C05443=1054.206,-122.391,-64.552,170.361,28.677,155.442
C05444=1054.213,-122.141,-64.561,170.364,28.677,155.442
C05445=1054.219,-121.892,-64.571,170.366,28.678,155.442
C05446=1054.225,-121.642,-64.580,170.368,28.678,155.442
C05447=1054.231,-121.393,-64.590,170.370,28.678,155.441
C05448=1054.237,-121.142,-64.598,170.371,28.679,155.441
C05449=1054.243,-120.892,-64.608,170.373,28.679,155.441
C05450=1054.249,-120.643,-64.618,170.376,28.680,155.441
C05451=1054.256,-120.393,-64.627,170.378,28.680,155.441
C05452=1054.263,-120.143,-64.636,170.380,28.681,155.441
C05453=1054.268,-119.894,-64.645,170.382,28.681,155.441
C05454=1054.274,-119.644,-64.655,170.384,28.682,155.441
C05455=1054.280,-119.394,-64.664,170.386,28.683,155.441
C05456=1054.286,-119.144,-64.673,170.389,28.683,155.441
C05457=1054.292,-118.894,-64.683,170.390,28.684,155.441
C05458=1054.299,-118.645,-64.692,170.392,28.684,155.441
C05459=1054.305,-118.395,-64.702,170.394,28.685,155.441
C05460=1054.311,-118.145,-64.712,170.396,28.685,155.440
C05461=1054.317,-117.896,-64.720,170.398,28.686,155.440
C05462=1054.323,-117.646,-64.730,170.401,28.686,155.440
C05463=1054.330,-117.397,-64.739,170.403,28.687,155.440
C05464=1054.336,-117.147,-64.749,170.405,28.688,155.440
C05465=1054.342,-116.897,-64.758,170.407,28.688,155.440
C05466=1054.348,-116.647,-64.768,170.409,28.689,155.440
C05467=1054.354,-116.397,-64.778,170.410,28.689,155.440
C05468=1054.360,-116.148,-64.787,170.412,28.689,155.440
C05469=1054.367,-115.898,-64.797,170.415,28.691,155.440
C05470=1054.373,-115.648,-64.806,170.417,28.691,155.440
C05471=1054.379,-115.364,-64.817,170.419,28.692,155.440
C05472=1054.387,-115.080,-64.828,170.422,28.692,155.440
C05473=1054.393,-114.795,-64.838,170.424,28.693,155.440
C05474=1054.401,-114.511,-64.850,170.427,28.694,155.439
C05475=1054.407,-114.261,-64.859,170.428,28.694,155.439
C05476=1054.413,-114.011,-64.869,170.430,28.695,155.439
C05477=1054.419,-113.762,-64.878,170.432,28.696,155.439
C05478=1054.425,-113.512,-64.887,170.434,28.696,155.439
C05479=1054.431,-113.263,-64.897,170.436,28.697,155.439
C05480=1054.437,-113.013,-64.908,170.439,28.698,155.439
C05481=1054.443,-112.763,-64.917,170.441,28.698,155.439
C05482=1054.449,-112.514,-64.927,170.443,28.699,155.439
C05483=1054.455,-112.264,-64.937,170.445,28.699,155.439
C05484=1054.462,-112.014,-64.946,170.446,28.700,155.439
C05485=1054.468,-111.764,-64.956,170.448,28.701,155.439
C05486=1054.474,-111.514,-64.965,170.450,28.702,155.439
C05487=1054.480,-111.265,-64.975,170.453,28.702,155.439
C05488=1054.487,-111.015,-64.985,170.455,28.703,155.439
C05489=1054.493,-110.766,-64.995,170.457,28.704,155.439
C05490=1054.498,-110.515,-65.005,170.459,28.704,155.439
C05491=1054.504,-110.266,-65.014,170.461,28.705,155.439
C05492=1054.511,-110.016,-65.024,170.462,28.706,155.439
C05493=1054.517,-109.766,-65.034,170.465,28.706,155.438
C05494=1054.523,-109.517,-65.044,170.467,28.707,155.438
C05495=1054.529,-109.267,-65.053,170.469,28.708,155.438
C05496=1054.535,-109.017,-65.063,170.471,28.708,155.438
C05497=1054.542,-108.768,-65.073,170.473,28.709,155.438
C05498=1054.548,-108.518,-65.083,170.475,28.710,155.438
C05499=1054.554,-108.268,-65.093,170.477,28.711,155.438
C05500=1054.560,-108.018,-65.103,170.479,28.711,155.438
C05501=1054.567,-107.768,-65.112,170.481,28.712,155.438
C05502=1054.573,-107.519,-65.123,170.483,28.713,155.438
C05503=1054.579,-107.269,-65.132,170.485,28.713,155.438
C05504=1054.585,-107.019,-65.142,170.487,28.714,155.438
C05505=1054.591,-106.769,-65.152,170.489,28.715,155.438
C05506=1054.597,-106.520,-65.162,170.491,28.716,155.438
C05507=1054.603,-106.270,-65.172,170.494,28.716,155.438
C05508=1054.610,-106.020,-65.181,170.495,28.717,155.438
C05509=1054.615,-105.771,-65.192,170.497,28.719,155.438
C05510=1054.622,-105.521,-65.202,170.499,28.719,155.438
C05511=1054.628,-105.271,-65.211,170.501,28.720,155.438
C05512=1054.634,-105.022,-65.222,170.503,28.720,155.438
C05513=1054.640,-104.772,-65.232,170.505,28.721,155.438
C05514=1054.646,-104.521,-65.242,170.508,28.722,155.438
C05515=1054.653,-104.272,-65.252,170.509,28.723,155.438
C05516=1054.658,-104.022,-65.262,170.511,28.724,155.438
C05517=1054.665,-103.773,-65.273,170.513,28.725,155.438
C05518=1054.671,-103.523,-65.282,170.515,28.726,155.438
C05519=1054.677,-103.273,-65.292,170.517,28.726,155.438
C05520=1054.683,-103.024,-65.303,170.519,28.727,155.438
C05521=1054.689,-102.774,-65.312,170.522,28.728,155.438
C05522=1054.695,-102.525,-65.322,170.523,28.729,155.438
C05523=1054.702,-102.274,-65.333,170.525,28.730,155.438
C05524=1054.708,-102.025,-65.343,170.527,28.731,155.438
C05525=1054.714,-101.775,-65.353,170.529,28.731,155.438
C05526=1054.720,-101.525,-65.363,170.531,28.732,155.438
C05527=1054.726,-101.276,-65.373,170.533,28.733,155.438
C05528=1054.732,-101.026,-65.383,170.536,28.734,155.437
C05529=1054.738,-100.777,-65.394,170.537,28.735,155.438
C05530=1054.745,-100.526,-65.404,170.539,28.736,155.438
C05531=1054.751,-100.277,-65.414,170.541,28.737,155.437
C05532=1054.757,-100.027,-65.424,170.543,28.738,155.437
C05533=1054.763,-99.778,-65.434,170.545,28.739,155.438
C05534=1054.769,-99.527,-65.445,170.547,28.739,155.437
C05535=1054.777,-99.242,-65.456,170.550,28.740,155.437
C05536=1054.784,-98.956,-65.468,170.551,28.741,155.437
C05537=1054.791,-98.670,-65.479,170.554,28.743,155.437
C05538=1054.798,-98.385,-65.492,170.556,28.744,155.437
C05539=1054.803,-98.135,-65.502,170.558,28.744,155.437
C05540=1054.810,-97.886,-65.512,170.560,28.745,155.437
C05541=1054.816,-97.636,-65.522,170.563,28.746,155.437
C05542=1054.822,-97.386,-65.533,170.564,28.747,155.437
C05543=1054.829,-97.137,-65.543,170.566,28.748,155.437
C05544=1054.834,-96.887,-65.553,170.568,28.749,155.437
C05545=1054.840,-96.637,-65.564,170.570,28.750,155.437
C05546=1054.847,-96.388,-65.575,170.572,28.751,155.437
C05547=1054.852,-96.138,-65.585,170.574,28.752,155.438
C05548=1054.859,-95.888,-65.595,170.575,28.753,155.438
C05549=1054.865,-95.638,-65.606,170.578,28.754,155.438
C05550=1054.871,-95.389,-65.616,170.580,28.755,155.438
C05551=1054.877,-95.139,-65.627,170.582,28.756,155.438
C05552=1054.882,-94.890,-65.638,170.584,28.757,155.438
C05553=1054.889,-94.639,-65.648,170.586,28.758,155.438
C05554=1054.895,-94.390,-65.658,170.587,28.759,155.438
C05555=1054.901,-94.140,-65.669,170.589,28.760,155.438
C05556=1054.907,-93.890,-65.679,170.591,28.761,155.438
C05557=1054.913,-93.641,-65.690,170.594,28.763,155.438
C05558=1054.920,-93.391,-65.700,170.596,28.763,155.438
C05559=1054.925,-93.141,-65.711,170.598,28.764,155.438
C05560=1054.932,-92.892,-65.721,170.600,28.765,155.438
C05561=1054.937,-92.642,-65.732,170.601,28.766,155.438
C05562=1054.944,-92.392,-65.743,170.603,28.767,155.438
C05563=1054.950,-92.143,-65.753,170.605,28.768,155.438
C05564=1054.956,-91.893,-65.763,170.607,28.769,155.438
C05565=1054.961,-91.643,-65.774,170.610,28.771,155.438
C05566=1054.968,-91.393,-65.785,170.611,28.772,155.438
C05567=1054.974,-91.144,-65.796,170.613,28.773,155.438
C05568=1054.981,-90.895,-65.806,170.615,28.774,155.438
C05569=1054.987,-90.644,-65.817,170.617,28.775,155.438
C05570=1054.992,-90.394,-65.827,170.619,28.776,155.438
C05571=1054.999,-90.145,-65.838,170.621,28.777,155.438
C05572=1055.005,-89.895,-65.849,170.622,28.778,155.438
C05573=1055.011,-89.645,-65.860,170.624,28.780,155.438
C05574=1055.017,-89.396,-65.870,170.627,28.781,155.438
C05575=1055.024,-89.146,-65.881,170.629,28.782,155.438
C05576=1055.029,-88.896,-65.892,170.631,28.783,155.438
C05577=1055.036,-88.647,-65.902,170.633,28.784,155.438
C05578=1055.041,-88.397,-65.913,170.634,28.785,155.438
C05579=1055.048,-88.147,-65.924,170.636,28.786,155.438
C05580=1055.054,-87.898,-65.934,170.638,28.787,155.438
C05581=1055.061,-87.648,-65.945,170.640,28.788,155.438
C05582=1055.066,-87.398,-65.956,170.643,28.789,155.438
C05583=1055.073,-87.149,-65.967,170.645,28.790,155.438
C05584=1055.079,-86.899,-65.978,170.646,28.791,155.439
C05585=1055.085,-86.649,-65.989,170.648,28.792,155.439
C05586=1055.091,-86.400,-65.999,170.650,28.794,155.439
C05587=1055.098,-86.150,-66.010,170.652,28.795,155.439
C05588=1055.103,-85.901,-66.021,170.654,28.796,155.439
C05589=1055.111,-85.651,-66.032,170.656,28.797,155.439
C05590=1055.116,-85.401,-66.043,170.657,28.798,155.439
C05591=1055.122,-85.152,-66.054,170.660,28.799,155.439
C05592=1055.129,-84.902,-66.064,170.662,28.800,155.439
C05593=1055.135,-84.652,-66.075,170.664,28.801,155.439
C05594=1055.141,-84.402,-66.086,170.666,28.803,155.439
C05595=1055.147,-84.153,-66.097,170.667,28.804,155.439
C05596=1055.153,-83.903,-66.108,170.669,28.805,155.439
C05597=1055.160,-83.653,-66.119,170.671,28.806,155.439
C05598=1055.165,-83.404,-66.130,170.673,28.807,155.439
C05599=1055.173,-83.120,-66.142,170.676,28.808,155.439
C05600=1055.180,-82.837,-66.154,170.678,28.810,155.439
C05601=1055.187,-82.553,-66.167,170.680,28.811,155.439
C05602=1055.194,-82.270,-66.179,170.682,28.812,155.439
C05603=1055.201,-82.020,-66.190,170.684,28.814,155.439
C05604=1055.206,-81.771,-66.201,170.686,28.815,155.440
C05605=1055.213,-81.521,-66.212,170.688,28.816,155.440
C05606=1055.219,-81.271,-66.223,170.689,28.817,155.440
C05607=1055.225,-81.021,-66.234,170.691,28.818,155.440
C05608=1055.231,-80.772,-66.245,170.694,28.820,155.440
C05609=1055.238,-80.522,-66.255,170.696,28.821,155.440
C05610=1055.244,-80.273,-66.267,170.698,28.822,155.440
C05611=1055.251,-80.023,-66.278,170.700,28.823,155.440
C05612=1055.256,-79.773,-66.289,170.701,28.825,155.440
C05613=1055.263,-79.523,-66.300,170.703,28.826,155.440
C05614=1055.269,-79.274,-66.311,170.705,28.827,155.440
C05615=1055.276,-79.024,-66.322,170.707,28.828,155.440
C05616=1055.282,-78.775,-66.334,170.709,28.829,155.440
C05617=1055.288,-78.525,-66.345,170.710,28.830,155.440
C05618=1055.294,-78.275,-66.356,170.713,28.832,155.440
C05619=1055.300,-78.025,-66.367,170.715,28.833,155.440
C05620=1055.306,-77.776,-66.378,170.717,28.835,155.441
C05621=1055.312,-77.526,-66.390,170.719,28.836,155.441
C05622=1055.318,-77.276,-66.401,170.720,28.837,155.441
C05623=1055.324,-77.026,-66.412,170.722,28.839,155.441
C05624=1055.331,-76.777,-66.423,170.724,28.840,155.441
C05625=1055.337,-76.527,-66.435,170.726,28.841,155.441
C05626=1055.343,-76.278,-66.446,170.728,28.842,155.441
C05627=1055.349,-76.027,-66.457,170.730,28.843,155.441
C05628=1055.355,-75.779,-66.468,170.731,28.845,155.441
C05629=1055.361,-75.528,-66.480,170.734,28.846,155.441
C05630=1055.367,-75.279,-66.491,170.736,28.848,155.441
C05631=1055.374,-75.029,-66.502,170.738,28.849,155.441
C05632=1055.379,-74.780,-66.513,170.739,28.851,155.441
C05633=1055.386,-74.530,-66.525,170.741,28.852,155.442
C05634=1055.392,-74.281,-66.536,170.743,28.853,155.442
C05635=1055.398,-74.031,-66.547,170.745,28.854,155.442
C05636=1055.405,-73.780,-66.559,170.747,28.856,155.442
C05637=1055.411,-73.532,-66.570,170.749,28.857,155.442
C05638=1055.417,-73.281,-66.582,170.750,28.859,155.442
C05639=1055.422,-73.032,-66.594,170.752,28.860,155.442
C05640=1055.429,-72.782,-66.605,170.754,28.861,155.442
C05641=1055.435,-72.533,-66.617,170.757,28.863,155.442
C05642=1055.441,-72.283,-66.628,170.758,28.864,155.442
C05643=1055.447,-72.033,-66.639,170.760,28.866,155.442
C05644=1055.453,-71.784,-66.651,170.762,28.867,155.443
C05645=1055.458,-71.534,-66.662,170.764,28.868,155.443
C05646=1055.465,-71.284,-66.674,170.766,28.870,155.443
C05647=1055.471,-71.035,-66.685,170.767,28.872,155.443
C05648=1055.477,-70.785,-66.697,170.769,28.873,155.443
C05649=1055.482,-70.536,-66.708,170.771,28.874,155.443
C05650=1055.489,-70.286,-66.720,170.773,28.876,155.443
C05651=1055.495,-70.036,-66.732,170.775,28.877,155.443
C05652=1055.501,-69.787,-66.744,170.776,28.879,155.443
C05653=1055.507,-69.536,-66.755,170.778,28.880,155.444
C05654=1055.513,-69.288,-66.767,170.780,28.881,155.444
C05655=1055.519,-69.037,-66.778,170.783,28.883,155.444
C05656=1055.525,-68.788,-66.790,170.784,28.885,155.444
C05657=1055.531,-68.538,-66.801,170.786,28.886,155.444
C05658=1055.538,-68.288,-66.813,170.788,28.887,155.444
C05659=1055.544,-68.040,-66.825,170.790,28.889,155.444
C05660=1055.549,-67.789,-66.837,170.792,28.891,155.444
C05661=1055.556,-67.540,-66.849,170.793,28.892,155.444
C05662=1055.562,-67.290,-66.859,170.795,28.893,155.445
C05663=1055.568,-67.009,-66.873,170.797,28.895,155.445
C05664=1055.576,-66.728,-66.886,170.800,28.897,155.445
C05665=1055.583,-66.446,-66.900,170.801,28.898,155.445
C05666=1055.590,-66.165,-66.913,170.803,28.900,155.445
C05667=1055.595,-65.915,-66.924,170.805,28.902,155.445
C05668=1055.602,-65.666,-66.936,170.807,28.903,155.445
C05669=1055.608,-65.416,-66.948,170.809,28.904,155.445
C05670=1055.614,-65.167,-66.959,170.810,28.906,155.446
C05671=1055.620,-64.917,-66.972,170.813,28.908,155.446
C05672=1055.626,-64.667,-66.984,170.815,28.909,155.446
C05673=1055.632,-64.418,-66.994,170.817,28.911,155.446
C05674=1055.638,-64.168,-67.007,170.819,28.912,155.446
C05675=1055.645,-63.918,-67.019,170.820,28.914,155.446
C05676=1055.651,-63.669,-67.030,170.822,28.915,155.446
C05677=1055.656,-63.419,-67.042,170.824,28.916,155.446
C05678=1055.663,-63.169,-67.054,170.826,28.918,155.447
C05679=1055.670,-62.920,-67.066,170.827,28.920,155.447
C05680=1055.675,-62.670,-67.078,170.829,28.921,155.447
C05681=1055.681,-62.421,-67.090,170.831,28.922,155.447
C05682=1055.688,-62.171,-67.102,170.833,28.924,155.447
C05683=1055.694,-61.921,-67.114,170.835,28.926,155.447
C05684=1055.700,-61.672,-67.125,170.836,28.927,155.447
C05685=1055.706,-61.422,-67.137,170.838,28.929,155.448
C05686=1055.713,-61.172,-67.149,170.840,28.930,155.448
C05687=1055.719,-60.923,-67.162,170.842,28.932,155.448
C05688=1055.725,-60.674,-67.173,170.844,28.933,155.448
C05689=1055.730,-60.423,-67.185,170.845,28.935,155.448
C05690=1055.737,-60.174,-67.197,170.848,28.937,155.448
C05691=1055.744,-59.924,-67.209,170.850,28.938,155.448
C05692=1055.749,-59.675,-67.221,170.852,28.939,155.448
C05693=1055.756,-59.425,-67.233,170.853,28.941,155.448
C05694=1055.762,-59.175,-67.244,170.855,28.943,155.449
C05695=1055.768,-58.925,-67.257,170.857,28.944,155.449
C05696=1055.775,-58.676,-67.269,170.859,28.946,155.449
C05697=1055.781,-58.427,-67.280,170.861,28.947,155.449
C05698=1055.787,-58.177,-67.293,170.862,28.949,155.449
C05699=1055.793,-57.927,-67.305,170.864,28.950,155.449
C05700=1055.800,-57.678,-67.317,170.866,28.952,155.449
C05701=1055.806,-57.428,-67.329,170.868,28.953,155.450
C05702=1055.812,-57.179,-67.341,170.869,28.955,155.450
C05703=1055.817,-56.928,-67.353,170.871,28.957,155.450
C05704=1055.824,-56.679,-67.365,170.873,28.958,155.450
C05705=1055.831,-56.429,-67.377,170.875,28.960,155.450
C05706=1055.837,-56.179,-67.389,170.877,28.961,155.450
C05707=1055.843,-55.930,-67.401,170.878,28.962,155.450
C05708=1055.850,-55.680,-67.413,170.880,28.964,155.450
C05709=1055.855,-55.431,-67.425,170.882,28.966,155.451
C05710=1055.862,-55.182,-67.437,170.884,28.967,155.451
C05711=1055.868,-54.932,-67.450,170.885,28.969,155.451
C05712=1055.874,-54.682,-67.462,170.887,28.971,155.451
C05713=1055.881,-54.433,-67.474,170.890,28.972,155.451
C05714=1055.887,-54.183,-67.486,170.892,28.974,155.451
C05715=1055.894,-53.933,-67.498,170.894,28.976,155.451
C05716=1055.900,-53.683,-67.511,170.895,28.977,155.452
C05717=1055.906,-53.434,-67.523,170.897,28.979,155.452
C05718=1055.913,-53.184,-67.535,170.899,28.981,155.452
C05719=1055.918,-52.935,-67.547,170.901,28.982,155.452
C05720=1055.925,-52.685,-67.559,170.902,28.983,155.452
C05721=1055.931,-52.435,-67.572,170.904,28.985,155.452
C05722=1055.937,-52.186,-67.584,170.906,28.986,155.452
C05723=1055.943,-51.936,-67.596,170.908,28.988,155.453
C05724=1055.950,-51.686,-67.608,170.910,28.990,155.453
C05725=1055.957,-51.437,-67.621,170.911,28.991,155.453
C05726=1055.963,-51.188,-67.633,170.913,28.993,155.453
C05727=1055.970,-50.907,-67.647,170.915,28.995,155.453
C05728=1055.977,-50.628,-67.661,170.918,28.997,155.453
C05729=1055.984,-50.347,-67.675,170.919,28.999,155.454
C05730=1055.990,-50.067,-67.688,170.921,29.000,155.454
C05731=1055.997,-49.818,-67.701,170.923,29.002,155.454
C05732=1056.003,-49.569,-67.714,170.925,29.004,155.454
C05733=1056.009,-49.319,-67.726,170.926,29.006,155.454
C05734=1056.016,-49.069,-67.738,170.928,29.007,155.454
C05735=1056.022,-48.819,-67.751,170.930,29.009,155.455
C05736=1056.027,-48.571,-67.764,170.932,29.011,155.455
C05737=1056.033,-48.321,-67.776,170.933,29.013,155.455
C05738=1056.040,-48.071,-67.788,170.935,29.014,155.455
C05739=1056.046,-47.821,-67.801,170.937,29.016,155.455
C05740=1056.052,-47.571,-67.813,170.939,29.018,155.455
C05741=1056.058,-47.322,-67.826,170.941,29.019,155.456
C05742=1056.065,-47.073,-67.838,170.942,29.021,155.456
C05743=1056.070,-46.823,-67.851,170.944,29.023,155.456
C05744=1056.076,-46.573,-67.863,170.946,29.025,155.456
C05745=1056.083,-46.324,-67.877,170.948,29.026,155.456
C05746=1056.089,-46.074,-67.889,170.949,29.028,155.456
C05747=1056.095,-45.824,-67.901,170.951,29.030,155.457
C05748=1056.101,-45.575,-67.915,170.953,29.032,155.457
C05749=1056.107,-45.325,-67.927,170.955,29.033,155.457
C05750=1056.114,-45.075,-67.939,170.956,29.035,155.457
C05751=1056.120,-44.826,-67.952,170.958,29.037,155.457
C05752=1056.126,-44.576,-67.965,170.960,29.039,155.458
C05753=1056.132,-44.326,-67.977,170.962,29.041,155.458
C05754=1056.138,-44.077,-67.991,170.963,29.042,155.458
C05755=1056.145,-43.828,-68.003,170.965,29.044,155.458
C05756=1056.151,-43.578,-68.015,170.967,29.046,155.458
C05757=1056.157,-43.328,-68.028,170.969,29.048,155.458
C05758=1056.163,-43.078,-68.041,170.970,29.049,155.459
C05759=1056.169,-42.829,-68.054,170.972,29.051,155.459
C05760=1056.176,-42.580,-68.066,170.974,29.053,155.459
C05761=1056.182,-42.330,-68.079,170.976,29.055,155.459
C05762=1056.188,-42.081,-68.092,170.978,29.056,155.459
C05763=1056.194,-41.831,-68.105,170.979,29.058,155.460
C05764=1056.200,-41.581,-68.117,170.981,29.060,155.460
C05765=1056.207,-41.332,-68.130,170.983,29.062,155.460
C05766=1056.212,-41.082,-68.142,170.984,29.064,155.460
C05767=1056.219,-40.833,-68.156,170.986,29.066,155.460
C05768=1056.225,-40.583,-68.168,170.988,29.067,155.461
C05769=1056.231,-40.334,-68.181,170.990,29.069,155.461
C05770=1056.237,-40.084,-68.193,170.992,29.071,155.461
C05771=1056.244,-39.835,-68.207,170.993,29.073,155.461
C05772=1056.250,-39.584,-68.220,170.995,29.074,155.461
C05773=1056.256,-39.335,-68.233,170.997,29.076,155.462
C05774=1056.262,-39.085,-68.245,170.999,29.078,155.462
C05775=1056.269,-38.836,-68.259,171.000,29.080,155.462
C05776=1056.275,-38.586,-68.271,171.002,29.082,155.462
C05777=1056.281,-38.337,-68.284,171.004,29.084,155.462
C05778=1056.287,-38.087,-68.297,171.006,29.085,155.462
C05779=1056.293,-37.837,-68.310,171.007,29.087,155.463
C05780=1056.299,-37.587,-68.323,171.009,29.089,155.463
C05781=1056.305,-37.338,-68.336,171.011,29.091,155.463
C05782=1056.311,-37.089,-68.349,171.013,29.093,155.463
C05783=1056.317,-36.839,-68.362,171.014,29.095,155.463
C05784=1056.324,-36.589,-68.376,171.016,29.097,155.464
C05785=1056.330,-36.339,-68.388,171.018,29.099,155.464
C05786=1056.336,-36.090,-68.401,171.020,29.100,155.464
C05787=1056.342,-35.841,-68.415,171.021,29.103,155.464
C05788=1056.348,-35.591,-68.427,171.023,29.104,155.464
C05789=1056.354,-35.342,-68.441,171.025,29.106,155.465
C05790=1056.360,-35.092,-68.453,171.026,29.108,155.465
C05791=1056.368,-34.812,-68.469,171.028,29.110,155.465
C05792=1056.374,-34.533,-68.483,171.030,29.112,155.465
C05793=1056.381,-34.253,-68.497,171.032,29.114,155.466
C05794=1056.388,-33.974,-68.513,171.033,29.116,155.466
C05795=1056.394,-33.724,-68.525,171.035,29.119,155.466
C05796=1056.400,-33.475,-68.539,171.037,29.120,155.466
C05797=1056.406,-33.226,-68.552,171.039,29.122,155.467
C05798=1056.413,-32.975,-68.565,171.040,29.124,155.467
C05799=1056.419,-32.726,-68.578,171.042,29.126,155.467
C05800=1056.425,-32.477,-68.591,171.044,29.128,155.467
C05801=1056.431,-32.227,-68.605,171.046,29.130,155.467
C05802=1056.437,-31.977,-68.617,171.047,29.132,155.468
C05803=1056.444,-31.728,-68.631,171.049,29.134,155.468
C05804=1056.450,-31.478,-68.644,171.051,29.135,155.468
C05805=1056.457,-31.229,-68.657,171.053,29.138,155.468
C05806=1056.462,-30.979,-68.671,171.054,29.139,155.468
C05807=1056.468,-30.729,-68.684,171.056,29.142,155.469
C05808=1056.474,-30.480,-68.697,171.058,29.143,155.469
C05809=1056.481,-30.230,-68.711,171.060,29.145,155.469
C05810=1056.487,-29.980,-68.723,171.061,29.147,155.469
C05811=1056.493,-29.731,-68.737,171.063,29.149,155.470
C05812=1056.499,-29.482,-68.750,171.064,29.151,155.470
C05813=1056.506,-29.232,-68.764,171.066,29.153,155.470
C05814=1056.512,-28.983,-68.777,171.068,29.154,155.470
C05815=1056.518,-28.733,-68.791,171.069,29.157,155.470
C05816=1056.524,-28.483,-68.803,171.071,29.158,155.471
C05817=1056.530,-28.234,-68.817,171.073,29.160,155.471
C05818=1056.537,-27.984,-68.830,171.075,29.162,155.471
C05819=1056.543,-27.735,-68.843,171.076,29.164,155.471
C05820=1056.549,-27.485,-68.857,171.078,29.166,155.472
C05821=1056.556,-27.235,-68.870,171.080,29.168,155.472
C05822=1056.562,-26.986,-68.884,171.081,29.170,155.472
C05823=1056.568,-26.737,-68.897,171.083,29.172,155.472
C05824=1056.574,-26.487,-68.911,171.085,29.174,155.472
C05825=1056.581,-26.237,-68.924,171.087,29.176,155.473
C05826=1056.586,-25.987,-68.938,171.088,29.178,155.473
C05827=1056.592,-25.738,-68.951,171.090,29.180,155.473
C05828=1056.598,-25.489,-68.964,171.092,29.182,155.473
C05829=1056.604,-25.238,-68.978,171.093,29.184,155.474
C05830=1056.611,-24.989,-68.992,171.094,29.186,155.474
C05831=1056.617,-24.740,-69.005,171.096,29.188,155.474
C05832=1056.622,-24.490,-69.019,171.098,29.190,155.474
C05833=1056.629,-24.240,-69.032,171.100,29.192,155.474
C05834=1056.635,-23.991,-69.046,171.101,29.194,155.475
C05835=1056.641,-23.741,-69.059,171.103,29.196,155.475
C05836=1056.647,-23.492,-69.073,171.105,29.198,155.475
C05837=1056.653,-23.242,-69.087,171.107,29.200,155.475
C05838=1056.659,-22.993,-69.100,171.108,29.202,155.476
C05839=1056.666,-22.744,-69.114,171.110,29.205,155.476
C05840=1056.672,-22.494,-69.128,171.112,29.206,155.476
C05841=1056.678,-22.244,-69.142,171.114,29.208,155.476
C05842=1056.684,-21.995,-69.155,171.115,29.211,155.477
C05843=1056.690,-21.745,-69.169,171.116,29.212,155.477
C05844=1056.697,-21.496,-69.182,171.118,29.214,155.477
C05845=1056.702,-21.246,-69.196,171.120,29.216,155.477
C05846=1056.709,-20.996,-69.210,171.121,29.219,155.478
C05847=1056.715,-20.747,-69.223,171.123,29.220,155.478
C05848=1056.721,-20.497,-69.237,171.125,29.222,155.478
C05849=1056.727,-20.247,-69.251,171.126,29.225,155.478
C05850=1056.733,-19.998,-69.265,171.128,29.227,155.479
C05851=1056.739,-19.749,-69.279,171.130,29.228,155.479
C05852=1056.746,-19.499,-69.292,171.132,29.231,155.479
C05853=1056.752,-19.249,-69.306,171.133,29.233,155.479
C05854=1056.758,-19.000,-69.319,171.135,29.235,155.480
C05855=1056.765,-18.720,-69.336,171.137,29.237,155.480
C05856=1056.772,-18.440,-69.351,171.139,29.239,155.480
C05857=1056.779,-18.159,-69.366,171.140,29.242,155.480
C05858=1056.786,-17.879,-69.382,171.142,29.244,155.481
C05859=1056.792,-17.630,-69.396,171.144,29.246,155.481
C05860=1056.798,-17.380,-69.409,171.146,29.248,155.481
C05861=1056.804,-17.130,-69.423,171.147,29.250,155.481
C05862=1056.811,-16.881,-69.437,171.149,29.252,155.482
C05863=1056.818,-16.631,-69.451,171.151,29.254,155.482
C05864=1056.823,-16.382,-69.465,171.153,29.256,155.482
C05865=1056.829,-16.133,-69.478,171.153,29.258,155.482
C05866=1056.836,-15.883,-69.493,171.155,29.260,155.483
C05867=1056.842,-15.634,-69.506,171.157,29.262,155.483
C05868=1056.848,-15.383,-69.520,171.158,29.264,155.483
C05869=1056.854,-15.134,-69.534,171.160,29.266,155.483
C05870=1056.861,-14.884,-69.549,171.162,29.268,155.484
C05871=1056.867,-14.635,-69.562,171.164,29.270,155.484
C05872=1056.872,-14.386,-69.576,171.165,29.273,155.484
C05873=1056.879,-14.136,-69.591,171.167,29.275,155.484
C05874=1056.885,-13.887,-69.604,171.169,29.277,155.485
C05875=1056.891,-13.636,-69.618,171.170,29.279,155.485
C05876=1056.897,-13.388,-69.632,171.171,29.281,155.485
C05877=1056.903,-13.138,-69.646,171.173,29.283,155.486
C05878=1056.909,-12.889,-69.661,171.175,29.285,155.486
C05879=1056.916,-12.639,-69.674,171.177,29.287,155.486
C05880=1056.922,-12.389,-69.688,171.178,29.289,155.486
C05881=1056.927,-12.140,-69.703,171.180,29.292,155.487
C05882=1056.934,-11.890,-69.717,171.182,29.294,155.487
C05883=1056.940,-11.641,-69.731,171.184,29.296,155.487
C05884=1056.946,-11.391,-69.746,171.184,29.298,155.487
C05885=1056.952,-11.142,-69.759,171.186,29.300,155.488
C05886=1056.958,-10.893,-69.773,171.188,29.302,155.488
C05887=1056.964,-10.642,-69.788,171.189,29.305,155.488
C05888=1056.971,-10.394,-69.802,171.191,29.307,155.488
C05889=1056.977,-10.143,-69.816,171.193,29.309,155.489
C05890=1056.983,-9.894,-69.830,171.195,29.311,155.489
C05891=1056.989,-9.644,-69.844,171.196,29.313,155.489
C05892=1056.995,-9.396,-69.859,171.197,29.315,155.489
C05893=1057.001,-9.145,-69.873,171.199,29.317,155.490
C05894=1057.008,-8.897,-69.887,171.201,29.319,155.490
C05895=1057.014,-8.646,-69.901,171.202,29.321,155.490
C05896=1057.020,-8.397,-69.916,171.204,29.324,155.491
C05897=1057.026,-8.147,-69.930,171.206,29.326,155.491
C05898=1057.032,-7.898,-69.944,171.208,29.328,155.491
C05899=1057.038,-7.648,-69.958,171.209,29.330,155.491
C05900=1057.045,-7.399,-69.973,171.210,29.332,155.492
C05901=1057.051,-7.149,-69.986,171.212,29.334,155.492
C05902=1057.057,-6.900,-70.001,171.214,29.337,155.492
C05903=1057.063,-6.650,-70.015,171.215,29.339,155.493
C05904=1057.070,-6.401,-70.029,171.217,29.341,155.493
C05905=1057.076,-6.152,-70.044,171.219,29.343,155.493
C05906=1057.082,-5.901,-70.058,171.220,29.345,155.493
C05907=1057.087,-5.652,-70.073,171.222,29.348,155.494
C05908=1057.094,-5.403,-70.086,171.223,29.350,155.494
C05909=1057.101,-5.153,-70.101,171.225,29.352,155.494
C05910=1057.106,-4.904,-70.116,171.226,29.353,155.494
C05911=1057.113,-4.654,-70.130,171.228,29.356,155.495
C05912=1057.119,-4.405,-70.144,171.230,29.358,155.495
C05913=1057.125,-4.155,-70.159,171.232,29.360,155.495
C05914=1057.131,-3.905,-70.173,171.233,29.362,155.495
C05915=1057.138,-3.656,-70.187,171.235,29.364,155.496
C05916=1057.144,-3.407,-70.202,171.236,29.366,155.496
C05917=1057.150,-3.157,-70.216,171.238,29.368,155.496
C05918=1057.156,-2.908,-70.231,171.239,29.371,155.497
C05919=1057.163,-2.625,-70.248,171.241,29.373,155.497
C05920=1057.169,-2.344,-70.264,171.243,29.376,155.497
C05921=1057.177,-2.062,-70.280,171.244,29.378,155.498
C05922=1057.184,-1.780,-70.297,171.246,29.381,155.498
C05923=1057.189,-1.531,-70.312,171.248,29.383,155.498
C05924=1057.196,-1.281,-70.326,171.250,29.386,155.499
C05925=1057.201,-1.032,-70.340,171.251,29.388,155.499
C05926=1057.208,-0.782,-70.355,171.253,29.390,155.499
C05927=1057.214,-0.532,-70.370,171.255,29.392,155.499
C05928=1057.220,-0.284,-70.385,171.256,29.395,155.500
C05929=1057.226,-0.033,-70.399,171.257,29.397,155.500
C05930=1057.232,0.216,-70.414,171.259,29.399,155.500
C05931=1057.238,0.465,-70.429,171.261,29.401,155.501
C05932=1057.244,0.715,-70.444,171.262,29.404,155.501
C05933=1057.250,0.964,-70.458,171.264,29.406,155.501
C05934=1057.257,1.214,-70.473,171.266,29.408,155.501
C05935=1057.262,1.463,-70.487,171.267,29.410,155.502
C05936=1057.268,1.713,-70.502,171.268,29.413,155.502
C05937=1057.274,1.963,-70.517,171.270,29.415,155.502
C05938=1057.280,2.212,-70.532,171.272,29.417,155.503
C05939=1057.286,2.461,-70.547,171.274,29.419,155.503
C05940=1057.293,2.711,-70.562,171.275,29.421,155.503
C05941=1057.298,2.960,-70.576,171.276,29.423,155.504
C05942=1057.305,3.210,-70.591,171.278,29.426,155.504
C05943=1057.311,3.460,-70.606,171.279,29.428,155.504
C05944=1057.317,3.709,-70.620,171.281,29.431,155.504
C05945=1057.323,3.959,-70.635,171.283,29.433,155.505
C05946=1057.329,4.208,-70.650,171.285,29.435,155.505
C05947=1057.335,4.457,-70.665,171.285,29.437,155.505
C05948=1057.342,4.707,-70.680,171.287,29.440,155.506
C05949=1057.348,4.957,-70.695,171.289,29.442,155.506
C05950=1057.354,5.205,-70.709,171.291,29.444,155.506
C05951=1057.360,5.455,-70.724,171.292,29.446,155.507
C05952=1057.366,5.705,-70.739,171.294,29.448,155.507
C05953=1057.372,5.954,-70.754,171.295,29.450,155.507
C05954=1057.378,6.204,-70.769,171.296,29.453,155.508
C05955=1057.384,6.453,-70.784,171.298,29.455,155.508
C05956=1057.391,6.703,-70.799,171.300,29.458,155.508
C05957=1057.396,6.952,-70.814,171.302,29.460,155.508
C05958=1057.403,7.202,-70.829,171.303,29.462,155.509
C05959=1057.409,7.451,-70.844,171.304,29.464,155.509
C05960=1057.415,7.700,-70.858,171.306,29.467,155.509
C05961=1057.421,7.950,-70.873,171.308,29.469,155.510
C05962=1057.428,8.200,-70.888,171.309,29.471,155.510
C05963=1057.434,8.449,-70.903,171.311,29.473,155.510
C05964=1057.440,8.698,-70.918,171.313,29.475,155.510
C05965=1057.446,8.948,-70.933,171.314,29.477,155.511
C05966=1057.452,9.198,-70.948,171.315,29.480,155.511
C05967=1057.459,9.447,-70.964,171.317,29.482,155.511
C05968=1057.465,9.696,-70.979,171.319,29.485,155.512
C05969=1057.471,9.945,-70.993,171.321,29.487,155.512
C05970=1057.477,10.195,-71.008,171.322,29.489,155.512
C05971=1057.484,10.445,-71.023,171.323,29.491,155.513
C05972=1057.490,10.694,-71.038,171.325,29.494,155.513
C05973=1057.495,10.944,-71.053,171.326,29.496,155.513
C05974=1057.501,11.193,-71.068,171.328,29.498,155.513
C05975=1057.508,11.442,-71.084,171.330,29.500,155.514
C05976=1057.514,11.692,-71.099,171.332,29.502,155.514
C05977=1057.521,11.942,-71.114,171.332,29.504,155.514
C05978=1057.527,12.191,-71.129,171.334,29.507,155.515
C05979=1057.533,12.440,-71.143,171.336,29.509,155.515
C05980=1057.539,12.690,-71.158,171.338,29.512,155.515
C05981=1057.545,12.939,-71.174,171.339,29.514,155.516
C05982=1057.552,13.189,-71.189,171.340,29.516,155.516
C05983=1057.559,13.472,-71.206,171.342,29.518,155.516
C05984=1057.566,13.756,-71.224,171.344,29.521,155.517
C05985=1057.573,14.041,-71.241,171.346,29.524,155.517
C05986=1057.580,14.324,-71.258,171.348,29.526,155.517
C05987=1057.587,14.573,-71.273,171.350,29.529,155.518
C05988=1057.592,14.823,-71.289,171.350,29.531,155.518
C05989=1057.599,15.073,-71.304,171.352,29.533,155.518
C05990=1057.604,15.322,-71.319,171.354,29.536,155.519
C05991=1057.610,15.571,-71.334,171.356,29.538,155.519
C05992=1057.617,15.821,-71.349,171.357,29.540,155.519
C05993=1057.623,16.070,-71.366,171.358,29.542,155.519
C05994=1057.629,16.320,-71.381,171.360,29.545,155.520
C05995=1057.636,16.570,-71.396,171.361,29.547,155.520
C05996=1057.641,16.818,-71.411,171.363,29.550,155.520
C05997=1057.647,17.068,-71.426,171.365,29.552,155.521
C05998=1057.653,17.318,-71.442,171.366,29.554,155.521
C05999=1057.660,17.567,-71.458,171.367,29.556,155.521
C06000=1057.666,17.817,-71.473,171.369,29.559,155.522
C06001=1057.672,18.067,-71.488,171.371,29.561,155.522
C06002=1057.678,18.316,-71.504,171.373,29.564,155.522
C06003=1057.684,18.565,-71.518,171.373,29.566,155.523
C06004=1057.690,18.814,-71.535,171.375,29.568,155.523
C06005=1057.697,19.064,-71.549,171.377,29.571,155.523
C06006=1057.702,19.313,-71.565,171.379,29.573,155.524
C06007=1057.709,19.563,-71.581,171.380,29.575,155.524
C06008=1057.715,19.812,-71.596,171.381,29.577,155.524
C06009=1057.721,20.062,-71.612,171.383,29.580,155.525
C06010=1057.728,20.311,-71.627,171.385,29.582,155.525
C06011=1057.734,20.561,-71.643,171.386,29.585,155.525
C06012=1057.739,20.809,-71.658,171.388,29.587,155.526
C06013=1057.745,21.059,-71.674,171.389,29.589,155.526
C06014=1057.752,21.308,-71.689,171.390,29.592,155.526
C06015=1057.758,21.558,-71.705,171.392,29.594,155.527
C06016=1057.764,21.807,-71.720,171.394,29.596,155.527
C06017=1057.770,22.057,-71.736,171.395,29.598,155.527
C06018=1057.776,22.307,-71.751,171.396,29.601,155.527
C06019=1057.782,22.556,-71.768,171.398,29.603,155.528
C06020=1057.789,22.806,-71.782,171.400,29.606,155.528
C06021=1057.795,23.055,-71.799,171.402,29.608,155.528
C06022=1057.800,23.305,-71.814,171.402,29.610,155.529
C06023=1057.807,23.554,-71.830,171.404,29.612,155.529
C06024=1057.812,23.803,-71.845,171.406,29.615,155.530
C06025=1057.819,24.052,-71.861,171.408,29.617,155.530
C06026=1057.825,24.302,-71.877,171.409,29.620,155.530
C06027=1057.831,24.551,-71.892,171.410,29.622,155.531
C06028=1057.837,24.801,-71.908,171.412,29.624,155.531
C06029=1057.843,25.050,-71.923,171.413,29.626,155.531
C06030=1057.849,25.300,-71.939,171.415,29.629,155.531
C06031=1057.856,25.549,-71.955,171.416,29.631,155.532
C06032=1057.862,25.799,-71.971,171.418,29.634,155.532
C06033=1057.868,26.048,-71.987,171.419,29.636,155.532
C06034=1057.874,26.298,-72.002,171.421,29.638,155.533
C06035=1057.880,26.547,-72.018,171.423,29.641,155.533
C06036=1057.887,26.796,-72.034,171.424,29.643,155.533
C06037=1057.892,27.046,-72.049,171.425,29.646,155.534
C06038=1057.898,27.295,-72.066,171.427,29.648,155.534
C06039=1057.905,27.544,-72.081,171.429,29.650,155.534
C06040=1057.910,27.794,-72.097,171.431,29.653,155.535
C06041=1057.917,28.043,-72.112,171.431,29.655,155.535
C06042=1057.923,28.293,-72.129,171.433,29.658,155.535
C06043=1057.929,28.542,-72.145,171.435,29.660,155.536
C06044=1057.935,28.792,-72.160,171.437,29.662,155.536
C06045=1057.941,29.041,-72.176,171.437,29.665,155.536
C06046=1057.947,29.290,-72.192,171.439,29.667,155.537
C06047=1057.954,29.576,-72.211,171.441,29.669,155.537
C06048=1057.962,29.861,-72.228,171.442,29.672,155.538
C06049=1057.968,30.145,-72.247,171.444,29.675,155.538
C06050=1057.975,30.431,-72.265,171.446,29.678,155.538
C06051=1057.981,30.680,-72.282,171.447,29.681,155.539
C06052=1057.987,30.930,-72.296,171.449,29.683,155.539
C06053=1057.993,31.179,-72.313,171.451,29.685,155.539
C06054=1057.999,31.429,-72.329,171.452,29.687,155.540
C06055=1058.005,31.678,-72.345,171.453,29.690,155.540
C06056=1058.012,31.927,-72.361,171.455,29.692,155.540
C06057=1058.018,32.176,-72.377,171.457,29.695,155.541
C06058=1058.024,32.427,-72.393,171.458,29.697,155.541
C06059=1058.030,32.676,-72.409,171.459,29.700,155.541
C06060=1058.036,32.926,-72.426,171.461,29.702,155.542
C06061=1058.043,33.175,-72.441,171.463,29.704,155.542
C06062=1058.049,33.424,-72.457,171.465,29.707,155.542
C06063=1058.055,33.673,-72.474,171.465,29.709,155.543
C06064=1058.061,33.923,-72.490,171.467,29.712,155.543
C06065=1058.066,34.172,-72.506,171.469,29.714,155.543
C06066=1058.073,34.422,-72.521,171.471,29.717,155.544
C06067=1058.079,34.671,-72.537,171.471,29.719,155.544
C06068=1058.085,34.920,-72.554,171.473,29.721,155.544
C06069=1058.091,35.170,-72.570,171.475,29.723,155.545
C06070=1058.097,35.419,-72.586,171.476,29.726,155.545
C06071=1058.104,35.669,-72.602,171.478,29.728,155.545
C06072=1058.110,35.918,-72.619,171.479,29.731,155.546
C06073=1058.116,36.168,-72.635,171.481,29.733,155.546
C06074=1058.122,36.417,-72.651,171.482,29.736,155.547
C06075=1058.128,36.666,-72.667,171.484,29.738,155.547
C06076=1058.134,36.915,-72.683,171.485,29.740,155.547
C06077=1058.140,37.165,-72.699,171.487,29.743,155.548
C06078=1058.146,37.414,-72.715,171.488,29.745,155.548
C06079=1058.153,37.664,-72.732,171.490,29.748,155.548
C06080=1058.159,37.913,-72.748,171.491,29.750,155.549
C06081=1058.165,38.163,-72.765,171.493,29.752,155.549
C06082=1058.171,38.412,-72.781,171.494,29.755,155.549
C06083=1058.177,38.661,-72.797,171.496,29.757,155.550
C06084=1058.183,38.911,-72.813,171.497,29.760,155.550
C06085=1058.189,39.160,-72.830,171.499,29.762,155.550
C06086=1058.195,39.409,-72.846,171.500,29.765,155.551
C06087=1058.201,39.660,-72.862,171.502,29.767,155.551
C06088=1058.207,39.908,-72.879,171.504,29.770,155.551
C06089=1058.213,40.158,-72.896,171.505,29.772,155.552
C06090=1058.219,40.407,-72.912,171.506,29.774,155.552
C06091=1058.225,40.656,-72.928,171.508,29.777,155.552
C06092=1058.231,40.906,-72.944,171.510,29.779,155.553
C06093=1058.237,41.155,-72.961,171.510,29.782,155.553
C06094=1058.244,41.405,-72.977,171.512,29.784,155.553
C06095=1058.250,41.654,-72.994,171.514,29.787,155.554
C06096=1058.256,41.903,-73.011,171.516,29.789,155.554
C06097=1058.262,42.152,-73.027,171.516,29.792,155.555
C06098=1058.268,42.402,-73.043,171.518,29.794,155.555
C06099=1058.274,42.651,-73.059,171.520,29.796,155.555
C06100=1058.280,42.901,-73.076,171.522,29.799,155.556
C06101=1058.286,43.151,-73.092,171.522,29.801,155.556
C06102=1058.293,43.399,-73.109,171.524,29.804,155.556
C06103=1058.299,43.693,-73.129,171.526,29.807,155.557
C06104=1058.306,43.986,-73.148,171.528,29.809,155.557
C06105=1058.313,44.279,-73.167,171.529,29.813,155.558
C06106=1058.320,44.572,-73.187,171.531,29.815,155.558
C06107=1058.326,44.817,-73.204,171.533,29.818,155.558
C06108=1058.332,45.062,-73.220,171.534,29.820,155.559
C06109=1058.337,45.308,-73.236,171.536,29.823,155.559
C06110=1058.344,45.554,-73.253,171.537,29.825,155.559
C06111=1058.349,45.799,-73.269,171.539,29.828,155.560
C06112=1058.355,46.044,-73.286,171.540,29.831,155.560
C06113=1058.361,46.289,-73.303,171.541,29.833,155.561
C06114=1058.366,46.535,-73.319,171.543,29.835,155.561
C06115=1058.372,46.784,-73.335,171.545,29.838,155.561
C06116=1058.379,47.034,-73.352,171.546,29.840,155.562
C06117=1058.384,47.283,-73.369,171.547,29.843,155.562
C06118=1058.391,47.532,-73.386,171.549,29.846,155.562
C06119=1058.397,47.782,-73.402,171.551,29.848,155.563
C06120=1058.403,48.032,-73.419,171.552,29.850,155.563
C06121=1058.409,48.281,-73.437,171.553,29.853,155.564
C06122=1058.415,48.530,-73.453,171.555,29.855,155.564
C06123=1058.421,48.779,-73.469,171.556,29.858,155.564
C06124=1058.426,49.028,-73.487,171.558,29.861,155.565
C06125=1058.433,49.278,-73.503,171.559,29.863,155.565
C06126=1058.439,49.527,-73.520,171.561,29.865,155.565
C06127=1058.445,49.776,-73.536,171.562,29.868,155.566
C06128=1058.450,50.026,-73.553,171.564,29.870,155.566
C06129=1058.457,50.276,-73.571,171.565,29.873,155.566
C06130=1058.463,50.525,-73.587,171.567,29.875,155.567
C06131=1058.469,50.774,-73.605,171.568,29.878,155.567
C06132=1058.475,51.024,-73.621,171.570,29.880,155.567
C06133=1058.481,51.273,-73.638,171.571,29.882,155.568
C06134=1058.487,51.522,-73.655,171.573,29.885,155.568
C06135=1058.493,51.771,-73.672,171.574,29.888,155.569
C06136=1058.499,52.021,-73.689,171.576,29.890,155.569
C06137=1058.505,52.270,-73.706,171.577,29.893,155.569
C06138=1058.511,52.520,-73.722,171.579,29.895,155.570
C06139=1058.518,52.769,-73.740,171.580,29.897,155.570
C06140=1058.523,53.019,-73.757,171.582,29.900,155.570
C06141=1058.529,53.267,-73.774,171.583,29.903,155.571
C06142=1058.536,53.517,-73.790,171.585,29.905,155.571
C06143=1058.541,53.766,-73.808,171.586,29.908,155.571
C06144=1058.547,54.016,-73.824,171.588,29.910,155.572
C06145=1058.554,54.265,-73.841,171.589,29.912,155.572
C06146=1058.559,54.515,-73.858,171.591,29.915,155.573
C06147=1058.565,54.764,-73.875,171.592,29.917,155.573
C06148=1058.572,55.013,-73.892,171.594,29.920,155.573
C06149=1058.578,55.263,-73.909,171.595,29.923,155.574
C06150=1058.584,55.511,-73.926,171.597,29.925,155.574
C06151=1058.590,55.762,-73.943,171.598,29.927,155.574
C06152=1058.596,56.011,-73.960,171.600,29.930,155.575
C06153=1058.602,56.259,-73.977,171.601,29.932,155.575
C06154=1058.608,56.510,-73.995,171.603,29.935,155.576
C06155=1058.614,56.758,-74.012,171.604,29.937,155.576
C06156=1058.621,57.008,-74.029,171.606,29.940,155.576
C06157=1058.626,57.257,-74.046,171.607,29.942,155.577
C06158=1058.633,57.506,-74.063,171.609,29.944,155.577
C06159=1058.639,57.756,-74.079,171.610,29.947,155.577
C06160=1058.645,58.005,-74.097,171.612,29.950,155.578
C06161=1058.651,58.255,-74.114,171.613,29.952,155.578
C06162=1058.657,58.504,-74.132,171.614,29.955,155.578
C06163=1058.663,58.753,-74.148,171.616,29.957,155.579
C06164=1058.670,59.003,-74.166,171.618,29.959,155.579
C06165=1058.675,59.252,-74.183,171.619,29.962,155.580
C06166=1058.682,59.502,-74.200,171.621,29.964,155.580
C06167=1058.687,59.751,-74.217,171.622,29.967,155.580
C06168=1058.694,60.000,-74.235,171.624,29.969,155.580
C06169=1058.700,60.249,-74.252,171.625,29.972,155.581
C06170=1058.706,60.499,-74.269,171.626,29.974,155.581
C06171=1058.713,60.748,-74.286,171.628,29.976,155.582
C06172=1058.718,60.997,-74.303,171.630,29.979,155.582
C06173=1058.725,61.246,-74.321,171.631,29.981,155.582
C06174=1058.731,61.496,-74.337,171.633,29.984,155.583
C06175=1058.738,61.781,-74.358,171.634,29.987,155.583
C06176=1058.745,62.066,-74.377,171.636,29.989,155.584
C06177=1058.752,62.351,-74.397,171.638,29.992,155.584
C06178=1058.759,62.635,-74.417,171.639,29.995,155.584
C06179=1058.766,62.885,-74.433,171.641,29.998,155.585
C06180=1058.771,63.134,-74.451,171.643,30.000,155.585
C06181=1058.778,63.383,-74.468,171.644,30.002,155.585
C06182=1058.784,63.632,-74.486,171.645,30.005,155.586
C06183=1058.791,63.882,-74.503,171.647,30.007,155.586
C06184=1058.796,64.131,-74.521,171.649,30.010,155.587
C06185=1058.803,64.380,-74.538,171.651,30.012,155.587
C06186=1058.808,64.630,-74.555,171.651,30.015,155.587
C06187=1058.815,64.879,-74.572,171.653,30.017,155.588
C06188=1058.821,65.128,-74.590,171.655,30.020,155.588
C06189=1058.827,65.378,-74.608,171.656,30.022,155.588
C06190=1058.833,65.627,-74.625,171.657,30.025,155.589
C06191=1058.839,65.876,-74.642,171.659,30.027,155.589
C06192=1058.845,66.126,-74.660,171.661,30.030,155.589
C06193=1058.851,66.374,-74.677,171.662,30.032,155.590
C06194=1058.857,66.624,-74.695,171.663,30.035,155.590
C06195=1058.863,66.873,-74.713,171.665,30.038,155.591
C06196=1058.869,67.123,-74.730,171.667,30.040,155.591
C06197=1058.876,67.372,-74.748,171.668,30.042,155.591
C06198=1058.881,67.621,-74.765,171.669,30.045,155.592
C06199=1058.887,67.871,-74.783,171.671,30.047,155.592
C06200=1058.893,68.120,-74.800,171.673,30.050,155.592
C06201=1058.900,68.370,-74.818,171.674,30.052,155.593
C06202=1058.905,68.619,-74.836,171.675,30.055,155.593
C06203=1058.912,68.868,-74.853,171.677,30.057,155.594
C06204=1058.917,69.117,-74.871,171.679,30.060,155.594
C06205=1058.924,69.367,-74.889,171.680,30.063,155.594
C06206=1058.929,69.616,-74.906,171.682,30.065,155.595
C06207=1058.936,69.865,-74.924,171.683,30.067,155.595
C06208=1058.941,70.114,-74.941,171.685,30.070,155.595
C06209=1058.948,70.364,-74.959,171.686,30.073,155.596
C06210=1058.953,70.613,-74.977,171.688,30.075,155.596
C06211=1058.960,70.862,-74.995,171.689,30.078,155.597
C06212=1058.965,71.111,-75.013,171.691,30.080,155.597
C06213=1058.972,71.361,-75.030,171.692,30.083,155.597
C06214=1058.978,71.610,-75.048,171.694,30.085,155.598
C06215=1058.984,71.859,-75.066,171.695,30.088,155.598
C06216=1058.990,72.109,-75.084,171.697,30.090,155.599
C06217=1058.995,72.358,-75.101,171.698,30.093,155.599
C06218=1059.002,72.607,-75.120,171.700,30.095,155.599
C06219=1059.007,72.856,-75.137,171.701,30.098,155.600
C06220=1059.014,73.106,-75.155,171.703,30.100,155.600
C06221=1059.020,73.356,-75.173,171.704,30.103,155.600
C06222=1059.026,73.605,-75.190,171.706,30.105,155.601
C06223=1059.032,73.854,-75.209,171.707,30.108,155.601
C06224=1059.038,74.103,-75.226,171.709,30.111,155.602
C06225=1059.044,74.353,-75.244,171.710,30.113,155.602
C06226=1059.049,74.602,-75.262,171.712,30.115,155.602
C06227=1059.055,74.851,-75.280,171.713,30.118,155.603
C06228=1059.062,75.100,-75.299,171.715,30.121,155.603
C06229=1059.067,75.349,-75.316,171.717,30.123,155.603
C06230=1059.074,75.599,-75.333,171.718,30.125,155.604
C06231=1059.080,75.849,-75.351,171.719,30.128,155.604
C06232=1059.086,76.097,-75.370,171.721,30.131,155.605
C06233=1059.092,76.347,-75.388,171.723,30.134,155.605
C06234=1059.098,76.596,-75.405,171.724,30.136,155.605
C06235=1059.104,76.845,-75.424,171.725,30.138,155.606
C06236=1059.110,77.095,-75.442,171.727,30.141,155.606
C06237=1059.116,77.344,-75.459,171.729,30.144,155.607
C06238=1059.122,77.593,-75.478,171.730,30.146,155.607
C06239=1059.129,77.877,-75.498,171.731,30.149,155.607
C06240=1059.136,78.163,-75.519,171.733,30.152,155.608
C06241=1059.143,78.447,-75.539,171.735,30.154,155.608
C06242=1059.150,78.731,-75.560,171.737,30.158,155.609
C06243=1059.156,78.981,-75.578,171.738,30.160,155.609
C06244=1059.161,79.230,-75.596,171.740,30.163,155.609
C06245=1059.168,79.479,-75.614,171.742,30.165,155.610
C06246=1059.173,79.729,-75.633,171.743,30.168,155.610
C06247=1059.179,79.978,-75.651,171.744,30.171,155.611
C06248=1059.185,80.227,-75.669,171.746,30.173,155.611
C06249=1059.191,80.477,-75.687,171.748,30.175,155.611
C06250=1059.197,80.726,-75.705,171.749,30.178,155.612
C06251=1059.203,80.975,-75.723,171.750,30.181,155.612
C06252=1059.210,81.224,-75.742,171.752,30.183,155.613
C06253=1059.214,81.474,-75.760,171.754,30.186,155.613
C06254=1059.221,81.723,-75.779,171.755,30.188,155.613
C06255=1059.227,81.973,-75.797,171.756,30.191,155.614
C06256=1059.233,82.221,-75.815,171.758,30.193,155.614
C06257=1059.239,82.471,-75.833,171.760,30.196,155.614
C06258=1059.245,82.720,-75.852,171.761,30.199,155.615
C06259=1059.250,82.969,-75.870,171.762,30.201,155.615
C06260=1059.257,83.218,-75.888,171.764,30.204,155.616
C06261=1059.263,83.468,-75.906,171.766,30.206,155.616
C06262=1059.269,83.717,-75.925,171.767,30.209,155.616
C06263=1059.275,83.966,-75.942,171.768,30.211,155.617
C06264=1059.281,84.215,-75.961,171.770,30.214,155.617
C06265=1059.286,84.465,-75.979,171.772,30.216,155.618
C06266=1059.292,84.714,-75.998,171.774,30.219,155.618
C06267=1059.299,84.963,-76.017,171.775,30.222,155.618
C06268=1059.305,85.213,-76.035,171.776,30.224,155.619
C06269=1059.311,85.461,-76.053,171.778,30.227,155.619
C06270=1059.316,85.711,-76.071,171.780,30.229,155.619
C06271=1059.322,85.960,-76.090,171.781,30.232,155.620
C06272=1059.329,86.210,-76.109,171.782,30.234,155.620
C06273=1059.334,86.459,-76.126,171.784,30.237,155.621
C06274=1059.341,86.708,-76.145,171.786,30.240,155.621
C06275=1059.347,86.957,-76.164,171.787,30.242,155.621
C06276=1059.353,87.207,-76.182,171.788,30.244,155.622
C06277=1059.359,87.456,-76.201,171.790,30.247,155.622
C06278=1059.365,87.705,-76.218,171.792,30.250,155.623
C06279=1059.371,87.954,-76.237,171.793,30.252,155.623
C06280=1059.377,88.204,-76.256,171.794,30.255,155.623
C06281=1059.383,88.453,-76.275,171.796,30.257,155.624
C06282=1059.389,88.702,-76.293,171.798,30.260,155.624
C06283=1059.395,88.951,-76.311,171.800,30.262,155.624
C06284=1059.401,89.200,-76.330,171.801,30.265,155.625
C06285=1059.407,89.450,-76.348,171.802,30.267,155.625
C06286=1059.413,89.699,-76.367,171.804,30.270,155.626
C06287=1059.420,89.948,-76.385,171.806,30.273,155.626
C06288=1059.426,90.197,-76.404,171.807,30.275,155.626
C06289=1059.431,90.447,-76.422,171.808,30.277,155.627
C06290=1059.437,90.696,-76.441,171.810,30.280,155.627
C06291=1059.444,90.945,-76.460,171.812,30.283,155.628
C06292=1059.449,91.194,-76.479,171.814,30.285,155.628
C06293=1059.455,91.443,-76.496,171.814,30.287,155.628
C06294=1059.461,91.693,-76.516,171.816,30.290,155.629
C06295=1059.467,91.942,-76.534,171.818,30.293,155.629
C06296=1059.473,92.191,-76.554,171.820,30.296,155.630
C06297=1059.479,92.441,-76.572,171.821,30.298,155.630
C06298=1059.484,92.689,-76.591,171.822,30.301,155.630
C06299=1059.490,92.939,-76.609,171.824,30.303,155.631
C06300=1059.496,93.188,-76.628,171.826,30.306,155.631
C06301=1059.503,93.438,-76.647,171.828,30.308,155.631
C06302=1059.509,93.687,-76.666,171.828,30.311,155.632
C06303=1059.515,93.971,-76.687,171.830,30.314,155.632
C06304=1059.522,94.256,-76.709,171.832,30.317,155.633
C06305=1059.529,94.540,-76.730,171.834,30.320,155.633
C06306=1059.536,94.826,-76.751,171.835,30.323,155.634
C06307=1059.542,95.075,-76.770,171.837,30.326,155.634
C06308=1059.548,95.324,-76.789,171.839,30.328,155.635
C06309=1059.553,95.573,-76.808,171.841,30.330,155.635
C06310=1059.559,95.822,-76.827,171.842,30.333,155.635
C06311=1059.566,96.071,-76.845,171.843,30.336,155.636
C06312=1059.571,96.321,-76.865,171.845,30.338,155.636
C06313=1059.578,96.570,-76.883,171.847,30.341,155.637
C06314=1059.583,96.819,-76.903,171.848,30.344,155.637
C06315=1059.590,97.068,-76.921,171.849,30.346,155.637
C06316=1059.596,97.318,-76.940,171.851,30.348,155.638
C06317=1059.601,97.566,-76.959,171.853,30.351,155.638
C06318=1059.607,97.815,-76.978,171.854,30.354,155.638
C06319=1059.613,98.065,-76.997,171.856,30.356,155.639
C06320=1059.619,98.314,-77.016,171.857,30.359,155.639
C06321=1059.625,98.563,-77.035,171.859,30.361,155.640
C06322=1059.631,98.813,-77.054,171.861,30.364,155.640
C06323=1059.637,99.062,-77.073,171.862,30.366,155.640
C06324=1059.643,99.311,-77.092,171.864,30.369,155.641
C06325=1059.649,99.561,-77.111,171.865,30.372,155.641
C06326=1059.655,99.810,-77.130,171.867,30.374,155.642
C06327=1059.661,100.059,-77.150,171.868,30.377,155.642
C06328=1059.668,100.308,-77.168,171.870,30.379,155.642
C06329=1059.674,100.557,-77.187,171.872,30.382,155.643
C06330=1059.680,100.806,-77.206,171.873,30.384,155.643
C06331=1059.686,101.056,-77.225,171.875,30.387,155.644
C06332=1059.691,101.305,-77.245,171.876,30.390,155.644
C06333=1059.696,101.554,-77.263,171.878,30.392,155.644
C06334=1059.703,101.803,-77.282,171.880,30.395,155.645
C06335=1059.709,102.052,-77.302,171.881,30.397,155.645
C06336=1059.715,102.301,-77.321,171.882,30.400,155.646
C06337=1059.720,102.551,-77.341,171.884,30.403,155.646
C06338=1059.727,102.800,-77.359,171.886,30.405,155.646
C06339=1059.732,103.049,-77.378,171.888,30.408,155.647
C06340=1059.738,103.298,-77.398,171.889,30.411,155.647
C06341=1059.744,103.547,-77.418,171.890,30.413,155.648
C06342=1059.751,103.797,-77.436,171.892,30.416,155.648
C06343=1059.756,104.046,-77.455,171.894,30.419,155.648
C06344=1059.762,104.295,-77.475,171.896,30.421,155.649
C06345=1059.768,104.544,-77.495,171.896,30.423,155.649
C06346=1059.774,104.793,-77.513,171.898,30.426,155.650
C06347=1059.780,105.043,-77.533,171.900,30.429,155.650
C06348=1059.786,105.292,-77.553,171.902,30.431,155.650
C06349=1059.792,105.541,-77.572,171.903,30.434,155.651
C06350=1059.797,105.790,-77.591,171.904,30.437,155.651
C06351=1059.804,106.040,-77.610,171.906,30.439,155.652
C06352=1059.810,106.288,-77.630,171.908,30.442,155.652
C06353=1059.815,106.538,-77.649,171.910,30.445,155.652
C06354=1059.821,106.787,-77.668,171.911,30.447,155.653
C06355=1059.827,107.036,-77.688,171.912,30.449,155.653
C06356=1059.834,107.285,-77.707,171.914,30.452,155.654
C06357=1059.839,107.535,-77.726,171.916,30.455,155.654
C06358=1059.845,107.783,-77.746,171.917,30.457,155.654
C06359=1059.851,108.033,-77.765,171.919,30.460,155.655
C06360=1059.857,108.282,-77.785,171.921,30.463,155.655
C06361=1059.863,108.531,-77.804,171.922,30.465,155.656
C06362=1059.869,108.780,-77.823,171.924,30.467,155.656
C06363=1059.875,109.029,-77.843,171.925,30.470,155.656
C06364=1059.881,109.278,-77.862,171.927,30.473,155.657
C06365=1059.887,109.527,-77.882,171.929,30.475,155.657
C06366=1059.893,109.776,-77.901,171.930,30.478,155.658
C06367=1059.899,110.062,-77.923,171.932,30.481,155.658
C06368=1059.906,110.346,-77.946,171.934,30.484,155.658
C06369=1059.913,110.631,-77.968,171.936,30.487,155.659
C06370=1059.920,110.915,-77.991,171.938,30.490,155.659
C06371=1059.927,111.165,-78.009,171.939,30.492,155.660
C06372=1059.933,111.413,-78.029,171.940,30.495,155.660
C06373=1059.938,111.663,-78.049,171.942,30.497,155.661
C06374=1059.944,111.912,-78.069,171.944,30.500,155.661
C06375=1059.950,112.161,-78.088,171.946,30.503,155.661
C06376=1059.956,112.410,-78.108,171.947,30.505,155.662
C06377=1059.962,112.659,-78.127,171.949,30.508,155.662
C06378=1059.968,112.909,-78.147,171.950,30.511,155.663
C06379=1059.974,113.158,-78.167,171.952,30.513,155.663
C06380=1059.980,113.407,-78.187,171.953,30.516,155.663
C06381=1059.986,113.656,-78.206,171.955,30.518,155.664
C06382=1059.992,113.905,-78.226,171.957,30.521,155.664
C06383=1059.998,114.154,-78.246,171.959,30.523,155.665
C06384=1060.004,114.404,-78.265,171.960,30.526,155.665
C06385=1060.009,114.653,-78.286,171.961,30.529,155.665
C06386=1060.014,114.902,-78.305,171.963,30.531,155.666
C06387=1060.020,115.151,-78.325,171.965,30.534,155.666
C06388=1060.026,115.400,-78.345,171.967,30.537,155.667
C06389=1060.033,115.650,-78.364,171.968,30.539,155.667
C06390=1060.038,115.899,-78.385,171.969,30.542,155.667
C06391=1060.044,116.148,-78.405,171.971,30.545,155.668
C06392=1060.050,116.397,-78.424,171.973,30.547,155.668
C06393=1060.056,116.646,-78.444,171.975,30.551,155.669
C06394=1060.062,116.895,-78.464,171.976,30.553,155.669
C06395=1060.067,117.144,-78.485,171.978,30.556,155.670
C06396=1060.073,117.393,-78.504,171.979,30.558,155.670
C06397=1060.079,117.642,-78.524,171.981,30.561,155.670
C06398=1060.085,117.891,-78.544,171.982,30.564,155.671
C06399=1060.090,118.141,-78.564,171.984,30.567,155.671
C06400=1060.096,118.390,-78.584,171.986,30.569,155.672
C06401=1060.102,118.639,-78.604,171.988,30.572,155.672
C06402=1060.108,118.888,-78.624,171.989,30.574,155.673
C06403=1060.114,119.137,-78.644,171.990,30.576,155.673
C06404=1060.119,119.386,-78.664,171.992,30.579,155.673
C06405=1060.125,119.635,-78.684,171.994,30.582,155.674
C06406=1060.132,119.885,-78.704,171.996,30.585,155.674
C06407=1060.138,120.134,-78.724,171.998,30.587,155.674
C06408=1060.143,120.383,-78.744,171.999,30.590,155.675
C06409=1060.149,120.632,-78.764,172.000,30.592,155.675
C06410=1060.155,120.881,-78.784,172.002,30.595,155.676
C06411=1060.161,121.130,-78.804,172.004,30.598,155.676
C06412=1060.166,121.380,-78.824,172.005,30.600,155.677
C06413=1060.172,121.628,-78.844,172.007,30.603,155.677
C06414=1060.178,121.877,-78.864,172.009,30.606,155.677
C06415=1060.184,122.127,-78.884,172.011,30.608,155.678
C06416=1060.190,122.377,-78.905,172.012,30.611,155.678
C06417=1060.196,122.625,-78.924,172.013,30.614,155.679
C06418=1060.202,122.874,-78.944,172.015,30.616,155.679
C06419=1060.208,123.123,-78.964,172.017,30.619,155.679
C06420=1060.214,123.373,-78.985,172.019,30.622,155.680
C06421=1060.220,123.622,-79.005,172.021,30.624,155.680
C06422=1060.226,123.870,-79.025,172.022,30.627,155.681
C06423=1060.231,124.120,-79.046,172.024,30.630,155.681
C06424=1060.238,124.369,-79.066,172.025,30.632,155.682
C06425=1060.244,124.618,-79.086,172.027,30.635,155.682
C06426=1060.250,124.867,-79.106,172.028,30.638,155.682
C06427=1060.255,125.116,-79.127,172.030,30.640,155.683
C06428=1060.261,125.365,-79.147,172.032,30.643,155.683
C06429=1060.267,125.614,-79.167,172.034,30.646,155.684
C06430=1060.273,125.863,-79.187,172.036,30.648,155.684
C06431=1060.280,126.148,-79.210,172.037,30.651,155.684
C06432=1060.286,126.432,-79.233,172.039,30.654,155.685
C06433=1060.293,126.717,-79.256,172.041,30.657,155.685
C06434=1060.300,127.002,-79.280,172.043,30.660,155.686
C06435=1060.306,127.251,-79.300,172.045,30.662,155.686
C06436=1060.312,127.500,-79.320,172.046,30.665,155.687
C06437=1060.318,127.749,-79.340,172.048,30.668,155.687
C06438=1060.324,127.998,-79.361,172.050,30.670,155.687
C06439=1060.330,128.247,-79.381,172.052,30.673,155.688
C06440=1060.336,128.496,-79.402,172.053,30.676,155.688
C06441=1060.342,128.745,-79.422,172.055,30.678,155.689
C06442=1060.348,128.994,-79.443,172.056,30.681,155.689
C06443=1060.354,129.244,-79.463,172.058,30.684,155.689
C06444=1060.360,129.493,-79.483,172.060,30.686,155.690
C06445=1060.366,129.742,-79.503,172.061,30.688,155.690
C06446=1060.372,129.991,-79.524,172.063,30.691,155.691
C06447=1060.378,130.240,-79.544,172.065,30.694,155.691
C06448=1060.384,130.489,-79.565,172.067,30.696,155.691
C06449=1060.390,130.738,-79.585,172.069,30.699,155.692
C06450=1060.396,130.987,-79.605,172.070,30.702,155.692
C06451=1060.402,131.237,-79.626,172.072,30.704,155.693
C06452=1060.408,131.485,-79.646,172.074,30.707,155.693
C06453=1060.414,131.734,-79.667,172.075,30.709,155.694
C06454=1060.420,131.984,-79.688,172.077,30.712,155.694
C06455=1060.426,132.233,-79.708,172.078,30.715,155.694
C06456=1060.432,132.481,-79.728,172.080,30.717,155.695
C06457=1060.438,132.731,-79.750,172.082,30.720,155.695
C06458=1060.444,132.979,-79.770,172.084,30.723,155.696
C06459=1060.450,133.229,-79.791,172.086,30.725,155.696
C06460=1060.455,133.478,-79.811,172.087,30.728,155.696
C06461=1060.461,133.727,-79.832,172.089,30.731,155.697
C06462=1060.467,133.976,-79.853,172.091,30.734,155.697
C06463=1060.473,134.225,-79.873,172.093,30.736,155.698
C06464=1060.479,134.474,-79.894,172.094,30.739,155.698
C06465=1060.484,134.724,-79.915,172.095,30.741,155.699
C06466=1060.490,134.972,-79.935,172.097,30.744,155.699
C06467=1060.497,135.222,-79.957,172.099,30.747,155.699
C06468=1060.503,135.470,-79.977,172.101,30.749,155.700
C06469=1060.508,135.720,-79.997,172.102,30.752,155.700
C06470=1060.514,135.969,-80.019,172.104,30.755,155.701
C06471=1060.520,136.218,-80.039,172.106,30.757,155.701
C06472=1060.526,136.467,-80.060,172.108,30.760,155.701
C06473=1060.531,136.716,-80.081,172.110,30.763,155.702
C06474=1060.538,136.965,-80.101,172.111,30.765,155.702
C06475=1060.544,137.214,-80.123,172.113,30.768,155.703
C06476=1060.549,137.463,-80.143,172.115,30.771,155.703
C06477=1060.556,137.712,-80.164,172.117,30.773,155.703
C06478=1060.561,137.961,-80.185,172.119,30.776,155.704
C06479=1060.567,138.210,-80.206,172.119,30.779,155.704
C06480=1060.573,138.459,-80.226,172.121,30.781,155.705
C06481=1060.579,138.708,-80.248,172.123,30.784,155.705
C06482=1060.584,138.957,-80.269,172.125,30.786,155.706
C06483=1060.591,139.207,-80.290,172.127,30.789,155.706
C06484=1060.597,139.455,-80.310,172.128,30.792,155.706
C06485=1060.603,139.705,-80.332,172.130,30.794,155.707
C06486=1060.608,139.954,-80.352,172.132,30.797,155.707
C06487=1060.614,140.203,-80.374,172.134,30.800,155.708
C06488=1060.620,140.452,-80.394,172.136,30.803,155.708
C06489=1060.626,140.700,-80.415,172.137,30.806,155.709
C06490=1060.632,140.950,-80.436,172.139,30.808,155.709
C06491=1060.637,141.199,-80.457,172.141,30.811,155.709
C06492=1060.643,141.448,-80.479,172.143,30.814,155.710
C06493=1060.649,141.697,-80.500,172.145,30.816,155.710
C06494=1060.655,141.946,-80.521,172.146,30.819,155.711
C06495=1060.661,142.230,-80.545,172.148,30.822,155.711
C06496=1060.668,142.515,-80.568,172.150,30.825,155.712
C06497=1060.675,142.800,-80.593,172.152,30.828,155.712
C06498=1060.682,143.084,-80.617,172.154,30.832,155.713
C06499=1060.688,143.332,-80.638,172.156,30.834,155.713
C06500=1060.693,143.582,-80.659,172.158,30.837,155.713
C06501=1060.699,143.830,-80.680,172.159,30.839,155.714
C06502=1060.705,144.080,-80.702,172.161,30.842,155.714
C06503=1060.711,144.328,-80.723,172.162,30.845,155.715
C06504=1060.717,144.578,-80.744,172.164,30.847,155.715
C06505=1060.723,144.827,-80.766,172.166,30.850,155.716
C06506=1060.729,145.075,-80.786,172.168,30.853,155.716
C06507=1060.735,145.325,-80.807,172.170,30.855,155.716
C06508=1060.740,145.574,-80.829,172.171,30.858,155.717
C06509=1060.747,145.823,-80.850,172.173,30.861,155.717
C06510=1060.752,146.071,-80.872,172.175,30.864,155.718
C06511=1060.758,146.321,-80.892,172.177,30.867,155.718
C06512=1060.764,146.571,-80.914,172.179,30.869,155.719
C06513=1060.770,146.819,-80.935,172.180,30.872,155.719
C06514=1060.776,147.068,-80.957,172.182,30.875,155.719
C06515=1060.781,147.317,-80.978,172.184,30.877,155.720
C06516=1060.787,147.567,-80.999,172.186,30.880,155.720
C06517=1060.793,147.816,-81.021,172.188,30.883,155.721
C06518=1060.799,148.064,-81.042,172.190,30.885,155.721
C06519=1060.805,148.313,-81.064,172.191,30.888,155.721
C06520=1060.811,148.562,-81.085,172.193,30.890,155.722
C06521=1060.817,148.811,-81.107,172.195,30.893,155.722
C06522=1060.822,149.060,-81.128,172.197,30.896,155.723
C06523=1060.828,149.310,-81.149,172.199,30.899,155.723
C06524=1060.834,149.559,-81.170,172.200,30.902,155.724
C06525=1060.840,149.807,-81.192,172.202,30.904,155.724
C06526=1060.846,150.056,-81.213,172.204,30.907,155.725
C06527=1060.852,150.305,-81.235,172.206,30.910,155.725
C06528=1060.858,150.554,-81.256,172.208,30.912,155.725
C06529=1060.864,150.803,-81.278,172.209,30.916,155.726
C06530=1060.869,151.052,-81.300,172.211,30.918,155.726
C06531=1060.875,151.301,-81.321,172.213,30.921,155.727
C06532=1060.881,151.551,-81.343,172.215,30.923,155.727
C06533=1060.887,151.799,-81.364,172.217,30.926,155.728
C06534=1060.893,152.048,-81.386,172.218,30.929,155.728
C06535=1060.899,152.297,-81.407,172.220,30.931,155.728
C06536=1060.904,152.546,-81.429,172.222,30.935,155.729
C06537=1060.910,152.795,-81.451,172.224,30.937,155.729
C06538=1060.916,153.044,-81.472,172.226,30.940,155.730
C06539=1060.922,153.293,-81.494,172.227,30.943,155.730
C06540=1060.928,153.542,-81.516,172.229,30.945,155.731
C06541=1060.934,153.791,-81.537,172.231,30.948,155.731
C06542=1060.939,154.040,-81.559,172.233,30.951,155.731
C06543=1060.945,154.290,-81.581,172.235,30.954,155.732
C06544=1060.951,154.538,-81.602,172.236,30.956,155.732
C06545=1060.957,154.787,-81.624,172.239,30.959,155.733
C06546=1060.963,155.036,-81.646,172.241,30.962,155.733
C06547=1060.969,155.285,-81.668,172.243,30.965,155.734
C06548=1060.974,155.534,-81.690,172.245,30.967,155.734
C06549=1060.980,155.783,-81.711,172.246,30.970,155.735
C06550=1060.987,156.032,-81.733,172.248,30.973,155.735
C06551=1060.991,156.281,-81.755,172.250,30.976,155.735
C06552=1060.998,156.530,-81.777,172.252,30.978,155.736
C06553=1061.004,156.779,-81.799,172.254,30.981,155.736
C06554=1061.009,157.028,-81.821,172.255,30.984,155.737
C06555=1061.015,157.277,-81.842,172.257,30.987,155.737
C06556=1061.021,157.526,-81.864,172.259,30.990,155.738
C06557=1061.028,157.775,-81.886,172.261,30.992,155.738
C06558=1061.033,158.024,-81.908,172.263,30.995,155.738
C06559=1061.040,158.308,-81.933,172.264,30.998,155.739
C06560=1061.046,158.592,-81.958,172.267,31.001,155.739
C06561=1061.053,158.877,-81.983,172.269,31.005,155.740
C06562=1061.060,159.160,-82.008,172.271,31.007,155.740
C06563=1061.065,159.409,-82.030,172.274,31.011,155.741
C06564=1061.072,159.659,-82.052,172.275,31.013,155.741
C06565=1061.078,159.907,-82.074,172.277,31.016,155.742
C06566=1061.083,160.156,-82.096,172.279,31.019,155.742
C06567=1061.089,160.405,-82.118,172.281,31.021,155.743
C06568=1061.095,160.655,-82.139,172.283,31.024,155.743
C06569=1061.100,160.903,-82.162,172.284,31.027,155.744
C06570=1061.107,161.152,-82.184,172.286,31.030,155.744
C06571=1061.112,161.401,-82.207,172.288,31.032,155.744
C06572=1061.118,161.650,-82.229,172.290,31.036,155.745
C06573=1061.123,161.899,-82.250,172.292,31.038,155.745
C06574=1061.129,162.148,-82.273,172.294,31.041,155.746
C06575=1061.134,162.397,-82.295,172.295,31.044,155.746
C06576=1061.140,162.645,-82.317,172.297,31.047,155.747
C06577=1061.146,162.895,-82.339,172.299,31.049,155.747
C06578=1061.151,163.144,-82.362,172.302,31.053,155.748
C06579=1061.158,163.393,-82.384,172.304,31.055,155.748
C06580=1061.163,163.641,-82.407,172.305,31.059,155.749
C06581=1061.168,163.890,-82.429,172.307,31.061,155.749
C06582=1061.175,164.139,-82.451,172.309,31.064,155.749
C06583=1061.180,164.389,-82.473,172.311,31.067,155.750
C06584=1061.185,164.637,-82.496,172.313,31.070,155.750
C06585=1061.191,164.886,-82.518,172.314,31.072,155.751
C06586=1061.197,165.135,-82.541,172.316,31.076,155.751
C06587=1061.203,165.384,-82.563,172.318,31.078,155.752
C06588=1061.208,165.633,-82.586,172.320,31.081,155.752
C06589=1061.214,165.881,-82.608,172.322,31.084,155.753
C06590=1061.220,166.131,-82.630,172.324,31.087,155.753
C06591=1061.225,166.380,-82.653,172.326,31.090,155.754
C06592=1061.231,166.629,-82.675,172.328,31.093,155.754
C06593=1061.237,166.878,-82.698,172.330,31.095,155.754
C06594=1061.242,167.126,-82.720,172.332,31.099,155.755
C06595=1061.248,167.375,-82.742,172.334,31.101,155.755
C06596=1061.254,167.624,-82.765,172.335,31.104,155.756
C06597=1061.260,167.873,-82.787,172.337,31.107,155.756
C06598=1061.265,168.122,-82.810,172.339,31.110,155.757
C06599=1061.271,168.371,-82.833,172.341,31.113,155.757
C06600=1061.277,168.620,-82.854,172.344,31.116,155.758
C06601=1061.282,168.869,-82.877,172.345,31.118,155.758
C06602=1061.288,169.118,-82.900,172.347,31.122,155.759
C06603=1061.294,169.366,-82.923,172.349,31.124,155.759
C06604=1061.300,169.616,-82.945,172.351,31.127,155.760
C06605=1061.306,169.865,-82.967,172.353,31.130,155.760
C06606=1061.311,170.113,-82.990,172.354,31.133,155.761
C06607=1061.317,170.362,-83.013,172.356,31.135,155.761
C06608=1061.323,170.612,-83.035,172.359,31.139,155.761
C06609=1061.329,170.860,-83.058,172.361,31.141,155.762
C06610=1061.335,171.109,-83.081,172.363,31.145,155.762
C06611=1061.340,171.358,-83.103,172.365,31.147,155.763
C06612=1061.346,171.607,-83.125,172.366,31.150,155.763
C06613=1061.352,171.856,-83.148,172.368,31.153,155.764
C06614=1061.358,172.105,-83.171,172.370,31.156,155.764
C06615=1061.363,172.353,-83.194,172.373,31.158,155.765
C06616=1061.370,172.602,-83.216,172.375,31.162,155.765
C06617=1061.375,172.851,-83.239,172.376,31.164,155.766
C06618=1061.381,173.100,-83.261,172.378,31.167,155.766
C06619=1061.387,173.349,-83.284,172.380,31.170,155.767
C06620=1061.392,173.598,-83.307,172.382,31.173,155.767
C06621=1061.399,173.847,-83.330,172.385,31.176,155.767
C06622=1061.405,174.096,-83.353,172.387,31.179,155.768
C06623=1061.411,174.379,-83.379,172.388,31.182,155.768
C06624=1061.418,174.663,-83.404,172.391,31.185,155.769
C06625=1061.424,174.947,-83.431,172.393,31.189,155.769
C06626=1061.431,175.231,-83.457,172.396,31.192,155.770
C06627=1061.437,175.480,-83.479,172.398,31.195,155.770
C06628=1061.443,175.729,-83.502,172.399,31.197,155.771
C06629=1061.449,175.978,-83.525,172.401,31.200,155.771
C06630=1061.454,176.226,-83.548,172.403,31.203,155.772
C06631=1061.460,176.475,-83.571,172.406,31.206,155.772
C06632=1061.466,176.724,-83.594,172.408,31.209,155.773
C06633=1061.472,176.973,-83.616,172.409,31.212,155.773
C06634=1061.478,177.222,-83.639,172.411,31.214,155.774
C06635=1061.484,177.471,-83.662,172.413,31.217,155.774
C06636=1061.490,177.720,-83.685,172.416,31.220,155.775
C06637=1061.495,177.968,-83.708,172.418,31.223,155.775
C06638=1061.502,178.218,-83.731,172.420,31.226,155.775
C06639=1061.508,178.467,-83.754,172.421,31.229,155.776
C06640=1061.514,178.715,-83.777,172.423,31.232,155.776
C06641=1061.520,178.964,-83.800,172.426,31.235,155.777
C06642=1061.526,179.213,-83.823,172.428,31.237,155.777
C06643=1061.531,179.462,-83.846,172.430,31.240,155.778
C06644=1061.537,179.710,-83.869,172.431,31.243,155.778
C06645=1061.543,179.959,-83.892,172.433,31.246,155.779
C06646=1061.550,180.209,-83.915,172.436,31.249,155.779
C06647=1061.556,180.458,-83.938,172.438,31.252,155.780
C06648=1061.562,180.706,-83.961,172.440,31.254,155.780
C06649=1061.567,180.955,-83.984,172.442,31.257,155.781
C06650=1061.573,181.204,-84.007,172.444,31.260,155.781
C06651=1061.579,181.453,-84.030,172.446,31.263,155.781
C06652=1061.585,181.701,-84.053,172.448,31.266,155.782
C06653=1061.591,181.951,-84.076,172.450,31.269,155.782
C06654=1061.597,182.199,-84.100,172.453,31.272,155.783
C06655=1061.603,182.448,-84.122,172.455,31.275,155.783
C06656=1061.609,182.697,-84.145,172.456,31.277,155.784
C06657=1061.615,182.946,-84.168,172.458,31.280,155.784
C06658=1061.621,183.195,-84.192,172.461,31.283,155.785
C06659=1061.627,183.444,-84.215,172.463,31.286,155.785
C06660=1061.633,183.692,-84.238,172.465,31.289,155.786
C06661=1061.639,183.941,-84.262,172.467,31.292,155.786
C06662=1061.645,184.190,-84.285,172.469,31.294,155.786
C06663=1061.651,184.439,-84.308,172.471,31.298,155.787
C06664=1061.657,184.688,-84.331,172.473,31.300,155.787
C06665=1061.663,184.936,-84.355,172.475,31.303,155.788
C06666=1061.668,185.186,-84.378,172.478,31.307,155.788
C06667=1061.674,185.434,-84.402,172.479,31.309,155.789
C06668=1061.680,185.683,-84.425,172.481,31.313,155.789
C06669=1061.685,185.932,-84.449,172.483,31.316,155.790
C06670=1061.691,186.181,-84.472,172.486,31.319,155.790
C06671=1061.696,186.430,-84.496,172.488,31.322,155.791
C06672=1061.702,186.678,-84.520,172.490,31.325,155.791
C06673=1061.708,186.927,-84.543,172.491,31.328,155.792
C06674=1061.713,187.176,-84.567,172.494,31.331,155.792
C06675=1061.719,187.425,-84.590,172.496,31.334,155.793
C06676=1061.726,187.674,-84.614,172.498,31.337,155.793
C06677=1061.731,187.923,-84.637,172.500,31.340,155.794
C06678=1061.737,188.171,-84.661,172.503,31.343,155.794
C06679=1061.742,188.420,-84.685,172.504,31.346,155.795
C06680=1061.748,188.669,-84.708,172.506,31.349,155.795
C06681=1061.754,188.917,-84.732,172.508,31.352,155.796
C06682=1061.759,189.167,-84.756,172.511,31.355,155.796
C06683=1061.765,189.415,-84.779,172.513,31.358,155.797
C06684=1061.770,189.664,-84.803,172.514,31.361,155.797
C06685=1061.776,189.913,-84.827,172.517,31.364,155.798
C06686=1061.782,190.163,-84.851,172.519,31.367,155.798
C06687=1061.789,190.445,-84.877,172.521,31.371,155.799
C06688=1061.796,190.729,-84.905,172.524,31.374,155.799
C06689=1061.801,191.012,-84.932,172.526,31.378,155.800
C06690=1061.809,191.295,-84.959,172.528,31.381,155.801
C06691=1061.814,191.544,-84.982,172.531,31.384,155.801
C06692=1061.820,191.793,-85.006,172.533,31.387,155.802
C06693=1061.825,192.041,-85.030,172.535,31.390,155.802
C06694=1061.832,192.290,-85.054,172.538,31.393,155.803
C06695=1061.838,192.539,-85.077,172.539,31.396,155.803
C06696=1061.843,192.788,-85.101,172.541,31.399,155.804
C06697=1061.849,193.036,-85.125,172.543,31.402,155.804
C06698=1061.855,193.286,-85.149,172.546,31.405,155.805
C06699=1061.861,193.534,-85.173,172.548,31.408,155.805
C06700=1061.866,193.783,-85.197,172.550,31.412,155.806
C06701=1061.873,194.032,-85.221,172.552,31.414,155.806
C06702=1061.878,194.280,-85.245,172.554,31.417,155.807
C06703=1061.884,194.529,-85.268,172.556,31.421,155.807
C06704=1061.890,194.779,-85.293,172.559,31.423,155.808
C06705=1061.896,195.027,-85.316,172.561,31.427,155.808
C06706=1061.901,195.275,-85.341,172.563,31.430,155.809
C06707=1061.908,195.524,-85.365,172.565,31.433,155.809
C06708=1061.912,195.774,-85.388,172.567,31.436,155.810
C06709=1061.919,196.023,-85.412,172.569,31.439,155.810
C06710=1061.925,196.271,-85.436,172.572,31.442,155.811
C06711=1061.930,196.519,-85.460,172.574,31.445,155.811
C06712=1061.937,196.768,-85.484,172.577,31.448,155.812
C06713=1061.942,197.017,-85.508,172.578,31.451,155.812
C06714=1061.949,197.266,-85.533,172.580,31.454,155.813
C06715=1061.954,197.515,-85.557,172.583,31.457,155.813
C06716=1061.960,197.763,-85.580,172.585,31.460,155.814
C06717=1061.966,198.012,-85.605,172.587,31.464,155.814
C06718=1061.972,198.260,-85.629,172.590,31.466,155.815
C06719=1061.978,198.510,-85.653,172.591,31.470,155.815
C06720=1061.984,198.758,-85.678,172.593,31.473,155.816
C06721=1061.990,199.007,-85.702,172.596,31.475,155.816
C06722=1061.995,199.256,-85.726,172.598,31.479,155.817
C06723=1062.001,199.504,-85.750,172.601,31.482,155.817
C06724=1062.007,199.753,-85.774,172.603,31.485,155.818
C06725=1062.013,200.002,-85.798,172.604,31.488,155.818
C06726=1062.019,200.251,-85.822,172.607,31.491,155.819
C06727=1062.025,200.499,-85.846,172.609,31.494,155.819
C06728=1062.031,200.749,-85.871,172.612,31.497,155.820
C06729=1062.037,200.997,-85.894,172.614,31.500,155.820
C06730=1062.043,201.246,-85.919,172.616,31.503,155.821
C06731=1062.049,201.494,-85.943,172.618,31.507,155.821
C06732=1062.055,201.744,-85.967,172.620,31.509,155.822
C06733=1062.060,201.992,-85.992,172.623,31.513,155.822
C06734=1062.067,202.241,-86.016,172.625,31.516,155.823
C06735=1062.073,202.489,-86.041,172.627,31.519,155.823
C06736=1062.079,202.739,-86.065,172.630,31.522,155.824
C06737=1062.084,202.987,-86.089,172.631,31.525,155.824
C06738=1062.090,203.236,-86.114,172.634,31.529,155.825
C06739=1062.096,203.485,-86.138,172.636,31.531,155.825
C06740=1062.102,203.733,-86.163,172.638,31.534,155.826
C06741=1062.107,203.982,-86.187,172.641,31.538,155.826
C06742=1062.113,204.231,-86.212,172.643,31.541,155.827
C06743=1062.119,204.480,-86.236,172.645,31.544,155.827
C06744=1062.125,204.728,-86.262,172.647,31.547,155.828
C06745=1062.131,204.977,-86.285,172.649,31.551,155.829
C06746=1062.137,205.226,-86.310,172.652,31.554,155.829
C06747=1062.142,205.474,-86.335,172.654,31.557,155.830
C06748=1062.148,205.723,-86.359,172.657,31.560,155.830
C06749=1062.153,205.972,-86.384,172.658,31.564,155.831
C06750=1062.160,206.221,-86.409,172.661,31.567,155.831
C06751=1062.185,207.269,-86.512,172.833,31.649,155.839
C06752=1062.190,207.495,-86.535,172.835,31.653,155.840
C06753=1062.196,207.722,-86.558,172.836,31.656,155.840
C06754=1062.201,207.947,-86.582,172.838,31.660,155.841
C06755=1062.207,208.173,-86.605,172.840,31.664,155.842
C06756=1062.212,208.400,-86.628,172.841,31.668,155.842
C06757=1062.218,208.626,-86.652,172.843,31.671,155.843
C06758=1062.223,208.853,-86.675,172.845,31.675,155.844
C06759=1062.229,209.079,-86.698,172.847,31.679,155.844
C06760=1062.236,209.327,-86.724,172.849,31.683,155.845
C06761=1062.241,209.576,-86.750,172.851,31.687,155.846
C06762=1062.247,209.825,-86.775,172.852,31.691,155.847
C06763=1062.253,210.074,-86.800,172.855,31.695,155.847
C06764=1062.260,210.322,-86.826,172.857,31.699,155.848
C06765=1062.266,210.570,-86.851,172.859,31.703,155.849
C06766=1062.271,210.819,-86.877,172.861,31.707,155.849
C06767=1062.277,211.067,-86.903,172.863,31.711,155.850
C06768=1062.283,211.316,-86.928,172.864,31.715,155.851
C06769=1062.289,211.565,-86.954,172.866,31.719,155.852
C06770=1062.295,211.813,-86.980,172.868,31.723,155.852
C06771=1062.302,212.062,-87.005,172.871,31.728,155.853
C06772=1062.308,212.311,-87.031,172.873,31.731,155.854
C06773=1062.314,212.559,-87.058,172.875,31.736,155.855
C06774=1062.320,212.808,-87.083,172.876,31.739,155.855
C06775=1062.326,213.057,-87.109,172.878,31.744,155.856
C06776=1062.332,213.306,-87.134,172.880,31.748,155.857
C06777=1062.338,213.554,-87.161,172.883,31.752,155.858
C06778=1062.344,213.803,-87.186,172.885,31.756,155.858
C06779=1062.351,214.051,-87.212,172.887,31.760,155.859
C06780=1062.356,214.300,-87.238,172.888,31.764,155.860
C06781=1062.362,214.548,-87.263,172.890,31.768,155.860
C06782=1062.368,214.797,-87.290,172.892,31.772,155.861
C06783=1062.374,215.045,-87.315,172.894,31.776,155.862
C06784=1062.380,215.294,-87.342,172.897,31.780,155.863
C06785=1062.386,215.542,-87.367,172.899,31.784,155.863
C06786=1062.392,215.791,-87.394,172.901,31.788,155.864
C06787=1062.398,216.039,-87.419,172.902,31.792,155.865
C06788=1062.404,216.288,-87.445,172.904,31.796,155.866
C06789=1062.410,216.537,-87.471,172.906,31.800,155.866
C06790=1062.416,216.785,-87.497,172.909,31.804,155.867
C06791=1062.423,217.034,-87.524,172.911,31.808,155.868
C06792=1062.428,217.283,-87.550,172.913,31.812,155.869
C06793=1062.435,217.531,-87.576,172.914,31.816,155.869
C06794=1062.440,217.780,-87.602,172.916,31.820,155.870
C06795=1062.447,218.028,-87.628,172.919,31.825,155.871
C06796=1062.452,218.277,-87.654,172.921,31.828,155.871
C06797=1062.459,218.525,-87.680,172.923,31.832,155.872
C06798=1062.464,218.774,-87.706,172.925,31.836,155.873
C06799=1062.471,219.023,-87.732,172.927,31.840,155.874
C06800=1062.477,219.271,-87.759,172.929,31.844,155.874
C06801=1062.484,219.519,-87.785,172.931,31.848,155.875
C06802=1062.489,219.768,-87.811,172.933,31.852,155.876
C06803=1062.495,220.016,-87.837,172.935,31.856,155.877
C06804=1062.502,220.266,-87.864,172.937,31.860,155.877
C06805=1062.508,220.514,-87.889,172.940,31.864,155.878
C06806=1062.514,220.763,-87.916,172.941,31.868,155.879
C06807=1062.520,221.011,-87.942,172.943,31.872,155.879
C06808=1062.525,221.240,-87.966,172.945,31.876,155.880
C06809=1062.531,221.468,-87.990,172.947,31.879,155.881
C06810=1062.537,221.697,-88.014,172.949,31.883,155.881
C06811=1062.543,221.926,-88.039,172.951,31.887,155.882
C06812=1062.548,222.155,-88.063,172.953,31.891,155.883
C06813=1062.553,222.383,-88.088,172.955,31.894,155.883
C06814=1062.559,222.612,-88.112,172.956,31.898,155.884
C06815=1062.564,222.841,-88.136,172.958,31.902,155.885
C06816=1062.571,223.089,-88.162,172.961,31.905,155.885
C06817=1062.576,223.337,-88.189,172.963,31.910,155.886
C06818=1062.583,223.586,-88.216,172.965,31.913,155.887
C06819=1062.588,223.835,-88.242,172.967,31.918,155.888
C06820=1062.595,224.083,-88.268,172.970,31.922,155.888
C06821=1062.601,224.332,-88.294,172.971,31.926,155.889
C06822=1062.606,224.580,-88.321,172.973,31.929,155.890
C06823=1062.613,224.829,-88.348,172.975,31.933,155.891
C06824=1062.618,225.077,-88.375,172.978,31.938,155.891
C06825=1062.625,225.325,-88.401,172.980,31.941,155.892
C06826=1062.631,225.574,-88.427,172.982,31.946,155.893
C06827=1062.637,225.823,-88.454,172.984,31.949,155.893
C06828=1062.643,226.071,-88.481,172.986,31.954,155.894
C06829=1062.649,226.320,-88.508,172.988,31.957,155.895
C06830=1062.656,226.568,-88.534,172.990,31.961,155.896
C06831=1062.661,226.817,-88.560,172.992,31.965,155.896
C06832=1062.667,227.066,-88.587,172.995,31.969,155.897
C06833=1062.673,227.315,-88.614,172.997,31.973,155.898
C06834=1062.679,227.563,-88.640,172.999,31.977,155.899
C06835=1062.686,227.811,-88.667,173.002,31.981,155.899
C06836=1062.692,228.059,-88.694,173.003,31.985,155.900
C06837=1062.698,228.308,-88.721,173.005,31.989,155.901
C06838=1062.704,228.556,-88.747,173.007,31.993,155.901
C06839=1062.710,228.805,-88.774,173.010,31.997,155.902
C06840=1062.716,229.054,-88.801,173.012,32.001,155.903
C06841=1062.723,229.302,-88.827,173.014,32.005,155.904
C06842=1062.729,229.551,-88.854,173.017,32.009,155.904
C06843=1062.735,229.799,-88.881,173.019,32.012,155.905
C06844=1062.740,230.048,-88.907,173.020,32.017,155.906
C06845=1062.747,230.297,-88.934,173.022,32.020,155.906
C06846=1062.753,230.544,-88.962,173.025,32.025,155.907
C06847=1062.759,230.793,-88.988,173.027,32.028,155.908
C06848=1062.765,231.042,-89.015,173.029,32.033,155.909
C06849=1062.771,231.290,-89.042,173.032,32.036,155.909
C06850=1062.777,231.538,-89.069,173.034,32.040,155.910
C06851=1062.783,231.787,-89.096,173.036,32.044,155.911
C06852=1062.789,232.035,-89.123,173.038,32.048,155.911
C06853=1062.795,232.284,-89.150,173.040,32.052,155.912
C06854=1062.801,232.533,-89.177,173.042,32.056,155.913
C06855=1062.807,232.781,-89.205,173.045,32.060,155.914
C06856=1062.813,233.030,-89.232,173.047,32.064,155.914
C06857=1062.819,233.278,-89.258,173.049,32.068,155.915
C06858=1062.825,233.527,-89.286,173.051,32.072,155.916
C06859=1062.831,233.775,-89.313,173.054,32.076,155.917
C06860=1062.837,234.023,-89.339,173.055,32.080,155.917
C06861=1062.844,234.272,-89.367,173.057,32.084,155.918
C06862=1062.849,234.520,-89.394,173.060,32.088,155.919
C06863=1062.855,234.769,-89.422,173.062,32.092,155.919
C06864=1062.861,234.993,-89.446,173.064,32.095,155.920
C06865=1062.866,235.218,-89.471,173.066,32.099,155.921
C06866=1062.872,235.443,-89.495,173.068,32.102,155.921
C06867=1062.877,235.668,-89.520,173.071,32.106,155.922
C06868=1062.883,235.892,-89.544,173.073,32.110,155.923
C06869=1062.888,236.117,-89.569,173.074,32.113,155.923
C06870=1062.893,236.341,-89.594,173.076,32.117,155.924
C06871=1062.899,236.567,-89.619,173.078,32.120,155.925
C06872=1062.905,236.815,-89.645,173.080,32.124,155.925
C06873=1062.911,237.064,-89.674,173.083,32.128,155.926
C06874=1062.917,237.312,-89.700,173.085,32.132,155.927
C06875=1062.924,237.561,-89.728,173.087,32.136,155.928
C06876=1062.930,237.808,-89.755,173.090,32.140,155.928
C06877=1062.936,238.057,-89.782,173.092,32.144,155.929
C06878=1062.941,238.305,-89.810,173.094,32.148,155.930
C06879=1062.948,238.555,-89.837,173.096,32.152,155.930
C06880=1062.954,238.802,-89.865,173.098,32.156,155.931
C06881=1062.960,239.051,-89.892,173.101,32.160,155.932
C06882=1062.966,239.299,-89.920,173.103,32.163,155.933
C06883=1062.972,239.548,-89.947,173.105,32.168,155.933
C06884=1062.978,239.796,-89.974,173.108,32.171,155.934
C06885=1062.985,240.045,-90.002,173.110,32.175,155.935
C06886=1062.990,240.293,-90.030,173.113,32.179,155.936
C06887=1062.996,240.542,-90.057,173.115,32.183,155.936
C06888=1063.003,240.790,-90.084,173.116,32.187,155.937
C06889=1063.008,241.038,-90.112,173.119,32.191,155.938
C06890=1063.015,241.287,-90.139,173.121,32.195,155.938
C06891=1063.021,241.535,-90.167,173.124,32.199,155.939
C06892=1063.027,241.784,-90.195,173.126,32.203,155.940
C06893=1063.033,242.032,-90.223,173.128,32.206,155.940
C06894=1063.039,242.281,-90.250,173.131,32.210,155.941
C06895=1063.045,242.529,-90.278,173.133,32.215,155.942
C06896=1063.051,242.777,-90.305,173.136,32.218,155.943
C06897=1063.057,243.026,-90.334,173.137,32.223,155.943
C06898=1063.063,243.274,-90.361,173.139,32.226,155.944
C06899=1063.069,243.523,-90.389,173.142,32.230,155.945
C06900=1063.076,243.771,-90.416,173.144,32.234,155.946
C06901=1063.081,244.019,-90.444,173.147,32.238,155.946
C06902=1063.088,244.268,-90.472,173.149,32.242,155.947
C06903=1063.093,244.516,-90.500,173.151,32.246,155.948
C06904=1063.100,244.764,-90.528,173.154,32.250,155.948
C06905=1063.106,245.013,-90.556,173.156,32.254,155.949
C06906=1063.112,245.261,-90.583,173.159,32.258,155.950
C06907=1063.118,245.510,-90.612,173.161,32.262,155.951
C06908=1063.124,245.758,-90.639,173.163,32.266,155.951
C06909=1063.130,246.006,-90.667,173.165,32.269,155.952
C06910=1063.136,246.255,-90.695,173.167,32.274,155.953
C06911=1063.142,246.503,-90.723,173.170,32.277,155.953
C06912=1063.148,246.751,-90.751,173.172,32.282,155.954
C06913=1063.154,247.000,-90.780,173.175,32.285,155.955
C06914=1063.160,247.248,-90.807,173.177,32.290,155.956
C06915=1063.166,247.497,-90.835,173.180,32.293,155.956
C06916=1063.172,247.745,-90.864,173.182,32.298,155.957
C06917=1063.177,247.993,-90.892,173.185,32.301,155.958
C06918=1063.184,248.242,-90.919,173.187,32.305,155.959
C06919=1063.189,248.490,-90.947,173.188,32.309,155.959
C06920=1063.196,248.793,-90.982,173.191,32.314,155.960
C06921=1063.204,249.095,-91.016,173.194,32.319,155.961
C06922=1063.211,249.398,-91.051,173.197,32.323,155.962
C06923=1063.218,249.701,-91.086,173.200,32.328,155.963
C06924=1063.224,249.950,-91.114,173.203,32.333,155.964
C06925=1063.231,250.198,-91.142,173.205,32.336,155.964
C06926=1063.236,250.446,-91.170,173.208,32.341,155.965
C06927=1063.242,250.695,-91.198,173.210,32.344,155.966
C06928=1063.248,250.943,-91.227,173.213,32.349,155.967
C06929=1063.254,251.192,-91.255,173.214,32.352,155.967
C06930=1063.260,251.439,-91.283,173.217,32.356,155.968
C06931=1063.266,251.688,-91.311,173.219,32.360,155.969
C06932=1063.272,251.936,-91.340,173.222,32.364,155.969
C06933=1063.278,252.185,-91.368,173.224,32.368,155.970
C06934=1063.284,252.433,-91.396,173.227,32.372,155.971
C06935=1063.291,252.681,-91.425,173.229,32.376,155.972
C06936=1063.297,252.930,-91.453,173.232,32.380,155.972
C06937=1063.303,253.178,-91.481,173.234,32.384,155.973
C06938=1063.308,253.426,-91.510,173.237,32.388,155.974
C06939=1063.314,253.675,-91.538,173.239,32.392,155.975
C06940=1063.320,253.923,-91.567,173.242,32.395,155.975
C06941=1063.327,254.171,-91.595,173.244,32.400,155.976
C06942=1063.333,254.420,-91.623,173.246,32.403,155.977
C06943=1063.339,254.667,-91.652,173.248,32.407,155.977
C06944=1063.345,254.916,-91.680,173.251,32.411,155.978
C06945=1063.351,255.164,-91.709,173.253,32.415,155.979
C06946=1063.357,255.413,-91.738,173.256,32.419,155.980
C06947=1063.364,255.661,-91.766,173.258,32.423,155.980
C06948=1063.370,255.910,-91.795,173.261,32.427,155.981
C06949=1063.376,256.158,-91.824,173.263,32.431,155.982
C06950=1063.381,256.406,-91.852,173.266,32.435,155.983
C06951=1063.388,256.654,-91.881,173.268,32.438,155.983
C06952=1063.394,256.903,-91.909,173.271,32.443,155.984
C06953=1063.400,257.151,-91.938,173.274,32.446,155.985
C06954=1063.406,257.399,-91.967,173.276,32.450,155.985
C06955=1063.413,257.647,-91.995,173.279,32.454,155.986
C06956=1063.419,257.895,-92.024,173.280,32.458,155.987
C06957=1063.425,258.144,-92.052,173.283,32.462,155.988
C06958=1063.431,258.392,-92.081,173.285,32.466,155.988
C06959=1063.437,258.640,-92.110,173.288,32.470,155.989
C06960=1063.443,258.889,-92.138,173.290,32.473,155.990
C06961=1063.450,259.137,-92.168,173.293,32.478,155.990
C06962=1063.456,259.386,-92.197,173.296,32.481,155.991
C06963=1063.461,259.634,-92.225,173.298,32.485,155.992
C06964=1063.471,260.022,-92.270,173.302,32.491,155.993
C06965=1063.481,260.411,-92.314,173.306,32.497,155.994
C06966=1063.491,260.799,-92.360,173.310,32.504,155.995
C06967=1063.501,261.188,-92.405,173.314,32.510,155.996
C06968=1063.507,261.436,-92.434,173.317,32.513,155.997
C06969=1063.513,261.684,-92.463,173.319,32.517,155.998
C06970=1063.519,261.933,-92.491,173.321,32.521,155.998
C06971=1063.525,262.181,-92.520,173.324,32.525,155.999
C06972=1063.532,262.401,-92.546,173.326,32.528,156.000
C06973=1063.537,262.622,-92.572,173.328,32.532,156.000
C06974=1063.542,262.842,-92.597,173.331,32.535,156.001
C06975=1063.548,263.063,-92.623,173.333,32.539,156.002
C06976=1063.553,263.284,-92.649,173.335,32.542,156.002
C06977=1063.560,263.504,-92.675,173.338,32.545,156.003
C06978=1063.565,263.724,-92.701,173.340,32.549,156.004
C06979=1063.570,263.945,-92.727,173.342,32.553,156.004
C06980=1063.576,264.193,-92.756,173.345,32.556,156.005
C06981=1063.582,264.442,-92.785,173.347,32.561,156.006
C06982=1063.588,264.690,-92.814,173.350,32.564,156.007
C06983=1063.594,264.938,-92.843,173.353,32.568,156.007
C06984=1063.600,265.186,-92.872,173.355,32.572,156.008
C06985=1063.606,265.434,-92.902,173.358,32.576,156.009
C06986=1063.613,265.682,-92.931,173.361,32.580,156.009
C06987=1063.618,265.930,-92.961,173.362,32.584,156.010
C06988=1063.625,266.179,-92.990,173.365,32.588,156.011
C06989=1063.631,266.427,-93.019,173.367,32.592,156.012
C06990=1063.637,266.675,-93.048,173.370,32.596,156.012
C06991=1063.643,266.923,-93.078,173.373,32.600,156.013
C06992=1063.649,267.171,-93.107,173.375,32.604,156.014
C06993=1063.655,267.419,-93.136,173.378,32.608,156.015
C06994=1063.661,267.669,-93.166,173.381,32.612,156.015
C06995=1063.668,267.916,-93.196,173.383,32.616,156.016
C06996=1063.674,268.164,-93.225,173.386,32.620,156.017
C06997=1063.680,268.413,-93.254,173.389,32.623,156.017
C06998=1063.686,268.661,-93.283,173.391,32.627,156.018
C06999=1063.692,268.909,-93.312,173.394,32.631,156.019
C07000=1063.698,269.157,-93.343,173.397,32.635,156.020
C07001=1063.704,269.405,-93.372,173.399,32.639,156.020
C07002=1063.710,269.653,-93.401,173.402,32.643,156.021
C07003=1063.717,269.902,-93.431,173.405,32.647,156.022
C07004=1063.723,270.150,-93.460,173.407,32.651,156.023
C07005=1063.729,270.398,-93.490,173.410,32.655,156.023
C07006=1063.735,270.646,-93.520,173.413,32.659,156.024
C07007=1063.741,270.894,-93.549,173.415,32.663,156.025
C07008=1063.747,271.142,-93.579,173.418,32.667,156.026
C07009=1063.753,271.391,-93.609,173.420,32.671,156.026
C07010=1063.760,271.639,-93.638,173.422,32.675,156.027
C07011=1063.765,271.887,-93.668,173.425,32.679,156.028
C07012=1063.772,272.135,-93.698,173.428,32.683,156.029
C07013=1063.778,272.383,-93.727,173.430,32.687,156.029
C07014=1063.784,272.631,-93.757,173.433,32.690,156.030
C07015=1063.791,272.880,-93.786,173.436,32.695,156.031
C07016=1063.796,273.127,-93.817,173.438,32.698,156.032
C07017=1063.802,273.376,-93.846,173.441,32.703,156.032
C07018=1063.808,273.623,-93.876,173.444,32.706,156.033
C07019=1063.814,273.872,-93.906,173.446,32.711,156.034
C07020=1063.821,274.120,-93.936,173.449,32.714,156.035
C07021=1063.827,274.369,-93.966,173.452,32.719,156.035
C07022=1063.832,274.616,-93.996,173.455,32.722,156.036
C07023=1063.839,274.864,-94.026,173.457,32.726,156.037
C07024=1063.845,275.113,-94.056,173.460,32.730,156.038
C07025=1063.851,275.361,-94.086,173.463,32.734,156.038
C07026=1063.857,275.609,-94.115,173.465,32.738,156.039
C07027=1063.863,275.857,-94.145,173.468,32.742,156.040
C07028=1063.869,276.080,-94.172,173.471,32.746,156.040
C07029=1063.874,276.301,-94.199,173.473,32.749,156.041
C07030=1063.880,276.524,-94.226,173.475,32.753,156.042
C07031=1063.886,276.746,-94.253,173.478,32.756,156.042
C07032=1063.890,276.969,-94.280,173.480,32.760,156.043
C07033=1063.896,277.191,-94.307,173.483,32.764,156.044
C07034=1063.902,277.413,-94.334,173.485,32.767,156.045
C07035=1063.907,277.635,-94.361,173.488,32.771,156.045
C07036=1063.913,277.884,-94.391,173.490,32.775,156.046
C07037=1063.919,278.132,-94.421,173.493,32.779,156.047
C07038=1063.926,278.379,-94.451,173.496,32.783,156.047
C07039=1063.932,278.628,-94.482,173.499,32.787,156.048
C07040=1063.938,278.876,-94.512,173.501,32.791,156.049
C07041=1063.944,279.124,-94.541,173.503,32.795,156.050
C07042=1063.950,279.372,-94.572,173.506,32.799,156.050
C07043=1063.956,279.620,-94.602,173.509,32.803,156.051
C07044=1063.962,279.868,-94.633,173.512,32.806,156.052
C07045=1063.969,280.116,-94.663,173.514,32.811,156.053
C07046=1063.975,280.364,-94.693,173.517,32.814,156.053
C07047=1063.981,280.613,-94.724,173.520,32.819,156.054
C07048=1063.987,280.860,-94.754,173.523,32.823,156.055
C07049=1063.993,281.108,-94.784,173.525,32.826,156.056
C07050=1064.000,281.357,-94.815,173.528,32.831,156.056
C07051=1064.005,281.605,-94.846,173.531,32.835,156.057
C07052=1064.011,281.852,-94.876,173.534,32.839,156.058
C07053=1064.018,282.101,-94.907,173.536,32.843,156.059
C07054=1064.023,282.349,-94.937,173.539,32.847,156.060
C07055=1064.029,282.597,-94.967,173.542,32.851,156.060
C07056=1064.036,282.845,-94.998,173.545,32.855,156.061
C07057=1064.041,283.093,-95.028,173.548,32.859,156.062
C07058=1064.048,283.341,-95.059,173.550,32.863,156.063
C07059=1064.054,283.589,-95.089,173.553,32.867,156.063
C07060=1064.060,283.837,-95.120,173.556,32.871,156.064
C07061=1064.067,284.085,-95.150,173.559,32.875,156.065
C07062=1064.073,284.332,-95.181,173.562,32.879,156.066
C07063=1064.079,284.581,-95.212,173.564,32.883,156.066
C07064=1064.085,284.829,-95.242,173.567,32.887,156.067
C07065=1064.091,285.077,-95.273,173.570,32.892,156.068
C07066=1064.097,285.325,-95.303,173.573,32.895,156.069
C07067=1064.104,285.573,-95.335,173.576,32.900,156.069
C07068=1064.110,285.821,-95.365,173.579,32.903,156.070
C07069=1064.116,286.069,-95.395,173.581,32.907,156.071
C07070=1064.122,286.317,-95.426,173.584,32.912,156.072
C07071=1064.129,286.565,-95.457,173.587,32.915,156.072
C07072=1064.135,286.813,-95.488,173.590,32.920,156.073
C07073=1064.141,287.061,-95.518,173.593,32.924,156.074
C07074=1064.147,287.309,-95.550,173.596,32.928,156.075
C07075=1064.154,287.557,-95.580,173.598,32.932,156.076
C07076=1064.159,287.805,-95.611,173.601,32.936,156.076
C07077=1064.165,288.053,-95.643,173.604,32.940,156.077
C07078=1064.171,288.301,-95.673,173.607,32.944,156.078
C07079=1064.178,288.550,-95.704,173.610,32.948,156.079
C07080=1064.184,288.797,-95.735,173.613,32.952,156.079
C07081=1064.190,289.045,-95.765,173.616,32.956,156.080
C07082=1064.196,289.292,-95.797,173.618,32.960,156.081
C07083=1064.203,289.541,-95.827,173.621,32.964,156.082
C07084=1064.208,289.768,-95.857,173.624,32.968,156.083
C07085=1064.214,289.996,-95.885,173.627,32.972,156.083
C07086=1064.219,290.223,-95.913,173.629,32.975,156.084
C07087=1064.225,290.451,-95.942,173.632,32.979,156.085
C07088=1064.231,290.679,-95.970,173.635,32.983,156.085
C07089=1064.237,290.907,-95.998,173.637,32.987,156.086
C07090=1064.242,291.134,-96.028,173.640,32.991,156.087
C07091=1064.248,291.362,-96.056,173.642,32.994,156.088
C07092=1064.254,291.609,-96.087,173.645,32.998,156.088
C07093=1064.260,291.858,-96.118,173.648,33.003,156.089
C07094=1064.266,292.105,-96.149,173.651,33.006,156.090
C07095=1064.272,292.353,-96.181,173.654,33.011,156.091
C07096=1064.279,292.602,-96.212,173.657,33.015,156.091
C07097=1064.285,292.849,-96.243,173.660,33.019,156.092
C07098=1064.291,293.097,-96.275,173.663,33.023,156.093
C07099=1064.297,293.346,-96.306,173.666,33.027,156.094
C07100=1064.303,293.593,-96.337,173.669,33.031,156.095
C07101=1064.310,293.841,-96.368,173.671,33.035,156.095
C07102=1064.316,294.089,-96.400,173.674,33.040,156.096
C07103=1064.322,294.337,-96.431,173.677,33.043,156.097
C07104=1064.329,294.585,-96.462,173.680,33.047,156.098
C07105=1064.335,294.833,-96.494,173.683,33.052,156.099
C07106=1064.341,295.080,-96.525,173.686,33.056,156.099
C07107=1064.347,295.328,-96.557,173.689,33.060,156.100
C07108=1064.353,295.577,-96.588,173.692,33.064,156.101
C07109=1064.359,295.824,-96.619,173.695,33.068,156.102
C07110=1064.365,296.072,-96.651,173.698,33.072,156.102
C07111=1064.372,296.320,-96.682,173.701,33.077,156.103
C07112=1064.377,296.568,-96.714,173.704,33.081,156.104
C07113=1064.384,296.816,-96.745,173.707,33.085,156.105
C07114=1064.390,297.064,-96.777,173.710,33.089,156.106
C07115=1064.397,297.312,-96.809,173.713,33.093,156.107
C07116=1064.402,297.559,-96.841,173.715,33.098,156.107
C07117=1064.408,297.807,-96.873,173.718,33.102,156.108
C07118=1064.415,298.055,-96.904,173.721,33.106,156.109
C07119=1064.420,298.303,-96.936,173.724,33.110,156.110
C07120=1064.426,298.551,-96.968,173.727,33.114,156.111
C07121=1064.433,298.799,-96.999,173.730,33.119,156.111
C07122=1064.438,299.046,-97.031,173.734,33.123,156.112
C07123=1064.444,299.295,-97.063,173.737,33.127,156.113
C07124=1064.451,299.542,-97.096,173.740,33.131,156.114
C07125=1064.457,299.790,-97.127,173.743,33.136,156.115
C07126=1064.463,300.038,-97.159,173.746,33.140,156.116
C07127=1064.469,300.286,-97.191,173.749,33.144,156.116
C07128=1064.475,300.534,-97.223,173.752,33.148,156.117
C07129=1064.481,300.782,-97.254,173.755,33.152,156.118
C07130=1064.487,301.029,-97.287,173.758,33.157,156.119
C07131=1064.493,301.277,-97.319,173.761,33.161,156.120
C07132=1064.499,301.525,-97.351,173.764,33.166,156.121
C07133=1064.506,301.773,-97.383,173.767,33.170,156.121
C07134=1064.512,302.021,-97.415,173.770,33.174,156.122
C07135=1064.517,302.268,-97.446,173.773,33.178,156.123
C07136=1064.523,302.517,-97.478,173.776,33.182,156.124
C07137=1064.530,302.764,-97.511,173.779,33.187,156.125
C07138=1064.536,303.012,-97.543,173.782,33.191,156.125
C07139=1064.542,303.260,-97.575,173.785,33.195,156.126
C07140=1064.549,303.495,-97.606,173.788,33.199,156.127
C07141=1064.554,303.730,-97.636,173.791,33.204,156.128
C07142=1064.560,303.965,-97.667,173.794,33.207,156.129
C07143=1064.566,304.200,-97.697,173.796,33.211,156.129
C07144=1064.572,304.435,-97.727,173.799,33.215,156.130
C07145=1064.578,304.670,-97.758,173.802,33.220,156.131
C07146=1064.584,304.906,-97.788,173.805,33.223,156.132
C07147=1064.590,305.141,-97.819,173.808,33.228,156.133
C07148=1064.596,305.388,-97.851,173.811,33.232,156.133
C07149=1064.602,305.636,-97.883,173.814,33.236,156.134
C07150=1064.608,305.884,-97.916,173.818,33.240,156.135
C07151=1064.614,306.132,-97.948,173.821,33.245,156.136
C07152=1064.621,306.380,-97.980,173.824,33.249,156.137
C07153=1064.627,306.627,-98.013,173.827,33.253,156.138
C07154=1064.633,306.875,-98.045,173.830,33.258,156.138
C07155=1064.640,307.123,-98.078,173.834,33.262,156.139
C07156=1064.646,307.371,-98.110,173.837,33.266,156.140
C07157=1064.652,307.619,-98.142,173.840,33.270,156.141
C07158=1064.659,307.866,-98.175,173.843,33.275,156.142
C07159=1064.665,308.114,-98.207,173.846,33.279,156.143
C07160=1064.671,308.362,-98.239,173.849,33.283,156.143
C07161=1064.678,308.609,-98.272,173.852,33.288,156.144
C07162=1064.684,308.858,-98.304,173.855,33.292,156.145
C07163=1064.690,309.105,-98.337,173.858,33.296,156.146
C07164=1064.696,309.353,-98.370,173.861,33.300,156.147
C07165=1064.702,309.600,-98.402,173.864,33.305,156.148
C07166=1064.709,309.848,-98.434,173.868,33.309,156.148
C07167=1064.715,310.096,-98.467,173.871,33.313,156.149
C07168=1064.722,310.344,-98.499,173.874,33.318,156.150
C07169=1064.729,310.592,-98.532,173.877,33.322,156.151
C07170=1064.735,310.839,-98.565,173.881,33.327,156.152
C07171=1064.741,311.088,-98.597,173.884,33.331,156.153
C07172=1064.747,311.335,-98.630,173.887,33.335,156.154
C07173=1064.754,311.583,-98.663,173.890,33.339,156.154
C07174=1064.760,311.830,-98.695,173.894,33.343,156.155
C07175=1064.766,312.078,-98.728,173.897,33.348,156.156
C07176=1064.773,312.326,-98.761,173.900,33.352,156.157
C07177=1064.780,312.574,-98.793,173.903,33.356,156.158
C07178=1064.786,312.821,-98.826,173.906,33.361,156.159
C07179=1064.793,313.069,-98.859,173.909,33.365,156.159
C07180=1064.799,313.316,-98.892,173.912,33.370,156.160
C07181=1064.806,313.565,-98.925,173.916,33.374,156.161
C07182=1064.812,313.812,-98.958,173.919,33.378,156.162
C07183=1064.818,314.060,-98.990,173.922,33.382,156.163
C07184=1064.824,314.308,-99.024,173.925,33.387,156.164
C07185=1064.830,314.555,-99.056,173.929,33.391,156.165
C07186=1064.836,314.804,-99.090,173.932,33.396,156.166
C07187=1064.843,315.052,-99.123,173.935,33.401,156.166
C07188=1064.849,315.299,-99.156,173.939,33.405,156.167
C07189=1064.855,315.546,-99.190,173.942,33.410,156.168
C07190=1064.861,315.794,-99.222,173.945,33.414,156.169
C07191=1064.867,316.042,-99.256,173.948,33.419,156.170
C07192=1064.873,316.289,-99.288,173.951,33.423,156.171
C07193=1064.880,316.537,-99.322,173.954,33.427,156.172
C07194=1064.886,316.785,-99.356,173.957,33.432,156.173
C07195=1064.892,317.033,-99.388,173.961,33.436,156.174
C07196=1064.898,317.270,-99.421,173.964,33.441,156.174
C07197=1064.904,317.507,-99.452,173.967,33.445,156.175
C07198=1064.909,317.744,-99.485,173.971,33.449,156.176
C07199=1064.916,317.981,-99.516,173.974,33.454,156.177
C07200=1064.922,318.218,-99.548,173.977,33.458,156.178
C07201=1064.928,318.455,-99.580,173.980,33.463,156.179
C07202=1064.934,318.692,-99.612,173.983,33.467,156.180
C07203=1064.939,318.928,-99.644,173.986,33.471,156.181
C07204=1064.946,319.176,-99.677,173.989,33.476,156.181
C07205=1064.952,319.424,-99.711,173.992,33.480,156.182
C07206=1064.958,319.671,-99.744,173.996,33.485,156.183
C07207=1064.964,319.919,-99.778,173.999,33.489,156.184
C07208=1064.971,320.167,-99.811,174.002,33.494,156.185
C07209=1064.977,320.414,-99.845,174.006,33.498,156.186
C07210=1064.983,320.662,-99.878,174.009,33.503,156.187
C07211=1064.989,320.910,-99.912,174.013,33.508,156.188
C07212=1064.996,321.157,-99.945,174.016,33.512,156.189
C07213=1065.002,321.405,-99.980,174.019,33.517,156.190
C07214=1065.008,321.653,-100.012,174.022,33.521,156.190
C07215=1065.014,321.900,-100.046,174.026,33.526,156.191
C07216=1065.021,322.148,-100.080,174.029,33.530,156.192
C07217=1065.027,322.396,-100.113,174.032,33.535,156.193
C07218=1065.034,322.643,-100.147,174.035,33.540,156.194
C07219=1065.040,322.891,-100.181,174.040,33.544,156.195
C07220=1065.046,323.139,-100.215,174.043,33.549,156.196
C07221=1065.053,323.386,-100.249,174.046,33.553,156.197
C07222=1065.059,323.634,-100.283,174.049,33.558,156.198
C07223=1065.066,323.882,-100.316,174.053,33.562,156.199
C07224=1065.071,324.129,-100.350,174.056,33.567,156.200
C07225=1065.079,324.377,-100.384,174.059,33.572,156.201
C07226=1065.084,324.624,-100.418,174.062,33.576,156.202
C07227=1065.091,324.872,-100.451,174.066,33.581,156.202
C07228=1065.097,325.120,-100.485,174.069,33.585,156.203
C07229=1065.104,325.368,-100.519,174.073,33.590,156.204
C07230=1065.110,325.615,-100.553,174.077,33.595,156.205
C07231=1065.117,325.863,-100.587,174.080,33.599,156.206
C07232=1065.124,326.110,-100.621,174.083,33.604,156.207
C07233=1065.130,326.358,-100.655,174.086,33.608,156.208
C07234=1065.136,326.606,-100.689,174.090,33.613,156.209
C07235=1065.143,326.853,-100.722,174.093,33.618,156.210
C07236=1065.149,327.101,-100.757,174.096,33.623,156.211
C07237=1065.156,327.348,-100.790,174.101,33.627,156.212
C07238=1065.162,327.596,-100.824,174.104,33.632,156.213
C07239=1065.169,327.844,-100.859,174.107,33.637,156.214
C07240=1065.175,328.091,-100.892,174.111,33.641,156.214
C07241=1065.182,328.339,-100.927,174.114,33.646,156.215
C07242=1065.188,328.587,-100.961,174.117,33.650,156.216
C07243=1065.195,328.833,-100.995,174.121,33.655,156.217
C07244=1065.201,329.081,-101.030,174.124,33.660,156.218
C07245=1065.208,329.329,-101.064,174.128,33.664,156.219
C07246=1065.214,329.576,-101.098,174.132,33.669,156.220
C07247=1065.221,329.824,-101.132,174.135,33.674,156.221
C07248=1065.227,330.072,-101.166,174.139,33.679,156.222
C07249=1065.234,330.319,-101.200,174.142,33.683,156.223
C07250=1065.240,330.567,-101.234,174.145,33.688,156.224
C07251=1065.247,330.815,-101.269,174.149,33.693,156.225
C07252=1065.254,331.049,-101.301,174.152,33.697,156.226
C07253=1065.259,331.283,-101.334,174.156,33.702,156.227
C07254=1065.265,331.516,-101.367,174.159,33.706,156.228
C07255=1065.271,331.751,-101.399,174.162,33.711,156.229
C07256=1065.277,331.985,-101.432,174.166,33.715,156.230
C07257=1065.284,332.219,-101.465,174.169,33.720,156.230
C07258=1065.289,332.453,-101.498,174.172,33.725,156.231
C07259=1065.295,332.687,-101.530,174.175,33.729,156.232
C07260=1065.302,332.935,-101.565,174.179,33.734,156.233
C07261=1065.308,333.182,-101.599,174.183,33.739,156.234
C07262=1065.314,333.429,-101.634,174.186,33.744,156.235
C07263=1065.321,333.677,-101.669,174.190,33.749,156.236
C07264=1065.328,333.925,-101.704,174.193,33.753,156.237
C07265=1065.333,334.172,-101.738,174.196,33.758,156.238
C07266=1065.340,334.419,-101.773,174.200,33.763,156.239
